# B&R Automation Studio project MotionTestBenchMaster (part 39)

```iecst
xInductionSetupActive	:= TRUE;

CASE uiInductionSetupStep OF
	0:
		IF	VAR_Machine.iq_stParameter.i_uiAxisSelected >= CST_FillerSubModuleHmiStart AND
			VAR_Machine.iq_stParameter.i_uiAxisSelected <= CST_FillerSubModuleHmiStart + CST_LastFillerModuleAxis	THEN

			VAR_Machine.stFillerModule.iq_stParameters.i_uiAxisSelected
				:=	VAR_Machine.iq_stParameter.i_uiAxisSelected - CST_FillerSubModuleHmiStart;

			uiInductionSetupStep	:=	100;
		ELSIF VAR_Machine.iq_stParameter.i_uiAxisSelected >= CST_InletSubModuleHmiStart AND
			VAR_Machine.iq_stParameter.i_uiAxisSelected <= CST_InletSubModuleHmiStart + CST_LastInletModuleAxis THEN

			VAR_Machine.stInletModule.iq_stParameters.i_uiAxisSelected
				:=	VAR_Machine.iq_stParameter.i_uiAxisSelected - CST_InletSubModuleHmiStart;

			uiInductionSetupStep	:=	200;
		ELSIF 	VAR_Machine.iq_stParameter.i_uiAxisSelected >= CST_OutletSubModuleHmiStart AND
			VAR_Machine.iq_stParameter.i_uiAxisSelected <= CST_OutletSubModuleHmiStart + CST_LastOutletModuleAxis THEN

			VAR_Machine.stOutletModule.iq_stParameters.i_uiAxisSelected
				:=	VAR_Machine.iq_stParameter.i_uiAxisSelected - CST_OutletSubModuleHmiStart;

			uiInductionSetupStep	:=	300;
		END_IF

	100:(* Induction motor setup on Filler Module *)
		VAR_Machine.stFillerModule.iq_stCmd.i_xInductionSetup :=	TRUE;

		IF VAR_Machine.stFillerModule.iq_stStatus.q_xInductionSetupActive 	AND
			VAR_Machine.stFillerModule.iq_stStatus.q_xInductionSetupDone	THEN

			VAR_Machine.stFillerModule.iq_stCmd.i_xInductionSetup 			:=	FALSE;
			VAR_Machine.stFillerModule.iq_stParameters.i_uiAxisSelected		:=	CST_FirstFillerModuleAxis;
			uiInductionSetupStep	:=	150;
		END_IF

	150:
		IF NOT VAR_Machine.stFillerModule.iq_stStatus.q_xInductionSetupActive 	AND
			NOT VAR_Machine.stFillerModule.iq_stStatus.q_xInductionSetupDone	THEN
			uiInductionSetupStep	:=	400;
		END_IF

	200:(* Induction motor setup on Inlet Module *)
		VAR_Machine.stInletModule.iq_stCmd.i_xInductionSetup :=	TRUE;

		IF VAR_Machine.stInletModule.iq_stStatus.q_xInductionSetupActive	AND
			VAR_Machine.stInletModule.iq_stStatus.q_xInductionSetupDone	THEN

			VAR_Machine.stInletModule.iq_stCmd.i_xInductionSetup 			:=	FALSE;
			VAR_Machine.stInletModule.iq_stParameters.i_uiAxisSelected		:=	CST_FirstInletModuleAxis;
			uiInductionSetupStep	:=	250;
		END_IF

	250:
		IF NOT VAR_Machine.stInletModule.iq_stStatus.q_xInductionSetupActive 	AND
			NOT	VAR_Machine.stInletModule.iq_stStatus.q_xInductionSetupDone	THEN
			uiInductionSetupStep	:=	400;
		END_IF

	300:(* Induction motor setup on Outlet Module *)
		VAR_Machine.stOutletModule.iq_stCmd.i_xInductionSetup :=	TRUE;

		IF VAR_Machine.stOutletModule.iq_stStatus.q_xInductionSetupActive	AND
			VAR_Machine.stOutletModule.iq_stStatus.q_xInductionSetupDone	THEN

			VAR_Machine.stOutletModule.iq_stCmd.i_xInductionSetup 			:=	FALSE;
			VAR_Machine.stOutletModule.iq_stParameters.i_uiAxisSelected		:=	CST_FirstOutletModuleAxis;
			uiInductionSetupStep	:=	350;
		END_IF

	350:
		IF NOT VAR_Machine.stOutletModule.iq_stStatus.q_xInductionSetupActive	AND
			NOT	VAR_Machine.stOutletModule.iq_stStatus.q_xInductionSetupDone	THEN
			uiInductionSetupStep	:=	400;
		END_IF

	400:
		xInductionSetupDone := TRUE;
END_CASE
END_STEP
ENTRY_ACTION
uiInductionSetupStep	:=	0;
xInductionSetupDone	:=	FALSE;
END_ACTION
EXIT_ACTION
VAR_Machine.stFillerModule.iq_stCmd.i_xInductionSetup 			:=	FALSE;
VAR_Machine.stFillerModule.iq_stParameters.i_uiAxisSelected		:=	CST_FirstFillerModuleAxis;

VAR_Machine.stOutletModule.iq_stCmd.i_xInductionSetup			:=	FALSE;
VAR_Machine.stOutletModule.iq_stParameters.i_uiAxisSelected		:=	CST_FirstOutletModuleAxis;

VAR_Machine.stInletModule.iq_stCmd.i_xInductionSetup			:=	FALSE;
VAR_Machine.stInletModule.iq_stParameters.i_uiAxisSelected		:=	CST_FirstInletModuleAxis;
END_ACTION
TRANSITION FROM InductionSetup TO InductionSetupExit:=
NOT xInductionSetupMode
END_TRANSITION
STEP InductionSetupExit:
xExitStep				:= TRUE;
xInductionSetupDone		:= FALSE;
xInductionSetupActive	:= FALSE;
END_STEP
TRANSITION FROM InductionSetupExit TO ModeSelection:=
xExitStep
END_TRANSITION
(* @SFCISJUMP := 'ModeSelection' *)
TRANSITION FROM ModeSelection TO StepByStep:=
xStepByStepMode
END_TRANSITION
STEP StepByStep:
IF xReactionActive OR uiStepByStep = 140 THEN
	xStepByStepMode	:= FALSE;
END_IF

xStepByStepActive	:= TRUE;

CASE uiStepByStep OF
	0:
		VAR_Machine.stFillerModule.iq_stCmd.i_xAutoMode	:= TRUE;
		VAR_Machine.stInletModule.iq_stCmd.i_xAutoMode	:= VAR_Machine.stInletModule.iq_stStatus.q_xModuleReal;
		VAR_Machine.stOutletModule.iq_stCmd.i_xAutoMode	:= VAR_Machine.stOutletModule.iq_stStatus.q_xModuleReal;
		uiStepByStep	:=	40;

	40:
		IF VAR_Machine.stFillerModule.iq_stStatus.q_xAutoActive		AND
			(VAR_Machine.stInletModule.iq_stStatus.q_xAutoActive	OR NOT
			VAR_Machine.stInletModule.iq_stStatus.q_xModuleReal)	AND
			(VAR_Machine.stOutletModule.iq_stStatus.q_xAutoActive	OR NOT
			VAR_Machine.stOutletModule.iq_stStatus.q_xModuleReal)	THEN

			IF NOT VAR_Machine.stFillerModule.iq_stStatus.q_xSynchroWithOffset	AND
				NOT VAR_Machine.stInletModule.iq_stStatus.q_xSynchroWithOffset	AND
				NOT VAR_Machine.stOutletModule.iq_stStatus.q_xSynchroWithOffset	THEN

				VAR_Machine.stMasterModule.iq_stParameters.i_lrRephasingPosition :=
					FC_RephasingMachine(iq_astInletSubModuleAxis	:= VAR_Machine.stInletModule.iq_astSubModuleAxis,
										iq_astFillerSubModuleAxis	:= VAR_Machine.stFillerModule.iq_astSubModuleAxis,
										iq_astOutletSubModuleAxis	:= VAR_Machine.stOutletModule.iq_astSubModuleAxis);

				VAR_Machine.stFillerModule.iq_stParameters.i_lrRephasingPosition
						:=	VAR_Machine.stMasterModule.iq_stParameters.i_lrRephasingPosition;

				VAR_Machine.stOutletModule.iq_stParameters.i_lrRephasingPosition
						:=	VAR_Machine.stMasterModule.iq_stParameters.i_lrRephasingPosition;

				VAR_Machine.stInletModule.iq_stParameters.i_lrRephasingPosition
					:=	VAR_Machine.stMasterModule.iq_stParameters.i_lrRephasingPosition;

				uiStepByStep	:=	100;
			END_IF
		END_IF

	100:
		VAR_Machine.stMasterModule.iq_stCmd.i_xPositioning				:= TRUE;
		VAR_Machine.stMasterModule.iq_stCmd.i_xMasterRephasingRequest	:= TRUE;

		IF VAR_Machine.stMasterModule.iq_stStatus.q_xPositioningActive AND VAR_Machine.stMasterModule.iq_stStatus.q_xMasterRephased THEN
			VAR_Machine.stMasterModule.iq_stCmd.i_xMasterRephasingRequest	:= FALSE;
			uiStepByStep	:=	110;
		END_IF

	110:
		VAR_Machine.stFillerModule.iq_stCmd.i_xStart	:= TRUE;
		VAR_Machine.stInletModule.iq_stCmd.i_xStart		:= VAR_Machine.stInletModule.iq_stStatus.q_xModuleReal;
		VAR_Machine.stOutletModule.iq_stCmd.i_xStart	:= VAR_Machine.stOutletModule.iq_stStatus.q_xModuleReal;
		uiStepByStep	:=	120;

	120:
		IF VAR_Machine.stFillerModule.iq_stStatus.q_xRealAxesSynchronized		AND
			VAR_Machine.stFillerModule.iq_stStatus.q_xAutoActive				AND
			VAR_Machine.stFillerModule.iq_stStatus.q_xMasterRephased			AND

			((VAR_Machine.stInletModule.iq_stStatus.q_xRealAxesSynchronized		AND
			VAR_Machine.stInletModule.iq_stStatus.q_xMasterRephased				AND
			VAR_Machine.stInletModule.iq_stStatus.q_xAutoActive)				OR NOT
			VAR_Machine.stInletModule.iq_stStatus.q_xModuleReal)				AND

			((VAR_Machine.stOutletModule.iq_stStatus.q_xRealAxesSynchronized	AND
			VAR_Machine.stOutletModule.iq_stStatus.q_xMasterRephased			AND
			VAR_Machine.stOutletModule.iq_stStatus.q_xAutoActive)				OR NOT
			VAR_Machine.stOutletModule.iq_stStatus.q_xModuleReal)				THEN

			VAR_Machine.stMasterModule.iq_stParameters.i_rPositioningOffset
				:= LREAL_TO_REAL(FC_LongRealReminder((VAR_Machine.stMasterModule.iq_stParameters.i_rStopPosition	- VAR_Machine.stMasterModule.iq_astSubModuleAxis[CST_MachineMasterAxis].iq_stStatus.q_stMainAxisStatus.q_lrPosition), 360.0, 0));

			IF VAR_Machine.stMasterModule.iq_stParameters.i_rPositioningOffset > 180.0 THEN
				VAR_Machine.stMasterModule.iq_stParameters.i_rPositioningOffset	:= VAR_Machine.stMasterModule.iq_stParameters.i_rPositioningOffset + 360.0 * (MAX(1, VAR_Machine.iq_stParameter.i_uiNumberOfSteps) - 1);
			ELSE
				VAR_Machine.stMasterModule.iq_stParameters.i_rPositioningOffset	:= VAR_Machine.stMasterModule.iq_stParameters.i_rPositioningOffset + 360.0 * MAX(1, VAR_Machine.iq_stParameter.i_uiNumberOfSteps);
			END_IF

			VAR_Machine.stMasterModule.iq_stCmd.i_xStart	:= TRUE;
			uiStepByStep := 130;
		END_IF

	130:
		IF VAR_Machine.stMasterModule.iq_stStatus.q_xPositioningDone THEN
			VAR_Machine.stMasterModule.iq_stCmd.i_xStart := FALSE;
			uiStepByStep := 140;
		END_IF

	140:

		xStepByStepDone	:= TRUE;
END_CASE
END_STEP
ENTRY_ACTION
uiStepByStep	:= 0;
xStepByStepDone	:= FALSE;
END_ACTION
EXIT_ACTION
VAR_Machine.stFillerModule.iq_stCmd.i_xAutoMode			:= FALSE;
VAR_Machine.stOutletModule.iq_stCmd.i_xAutoMode			:= FALSE;
VAR_Machine.stInletModule.iq_stCmd.i_xAutoMode			:= FALSE;

VAR_Machine.stMasterModule.iq_stCmd.i_xPositioning				:= FALSE;
VAR_Machine.stMasterModule.iq_stCmd.i_xStart					:= FALSE;
VAR_Machine.stMasterModule.iq_stCmd.i_xMasterRephasingRequest	:= FALSE;

VAR_Machine.stFillerModule.iq_stCmd.i_xStart	:= FALSE;
VAR_Machine.stInletModule.iq_stCmd.i_xStart		:= FALSE;
VAR_Machine.stOutletModule.iq_stCmd.i_xStart	:= FALSE;
END_ACTION
TRANSITION FROM StepByStep TO StepExit:=
NOT xStepByStepMode
END_TRANSITION
STEP StepExit:
IF NOT VAR_Machine.stMasterModule.iq_stStatus.q_xPositioningActive	AND
	NOT VAR_Machine.stFillerModule.iq_stStatus.q_xAutoActive		AND

	(NOT VAR_Machine.stOutletModule.iq_stStatus.q_xAutoActive		OR NOT
	VAR_Machine.stOutletModule.iq_stStatus.q_xModuleReal)			AND

	(NOT VAR_Machine.stInletModule.iq_stStatus.q_xAutoActive		OR NOT
	VAR_Machine.stInletModule.iq_stStatus.q_xModuleReal)			AND

	VAR_Machine.iq_stStatus.q_xMachineStopped 						THEN

	xStepByStepDone		:= FALSE;
	xStepByStepActive	:= FALSE;
	xExitStep			:= TRUE;
END_IF
END_STEP
TRANSITION FROM StepExit TO ModeSelection:=
xExitStep
END_TRANSITION
(* @SFCISJUMP := 'ModeSelection' *)
TRANSITION FROM ModeSelection TO StepByStepSingleAxis:=
xStepByStepSingleAxisMode
END_TRANSITION
STEP StepByStepSingleAxis:
xReactionOnFillerModule		:= xReactFillerEmergencyStop 	OR xReactFillerQuickStop		OR xReactFillerStop;//V1.7.2

IF xReactionOnFillerModule OR uiStepByStepSingleAxis = 130 THEN//V1.7.2
	xStepByStepSingleAxisMode	:= FALSE;
END_IF

xStepByStepSingleAxisActive	:= TRUE;

CASE uiStepByStepSingleAxis OF//V4.A.A.1.7.0
	0:
		IF	VAR_Machine.iq_stParameter.i_uiAxisSelected >= CST_FillerSubModuleHmiStart AND
			VAR_Machine.iq_stParameter.i_uiAxisSelected <= CST_FillerSubModuleHmiStart + CST_LastFillerModuleAxis	THEN

			VAR_Machine.stFillerModule.iq_stParameters.i_uiAxisSelected := VAR_Machine.iq_stParameter.i_uiAxisSelected - CST_FillerSubModuleHmiStart;

			uiStepByStepSingleAxis	:=	100;//Filler Module
		ELSIF VAR_Machine.iq_stParameter.i_uiAxisSelected >= CST_InletSubModuleHmiStart AND
			VAR_Machine.iq_stParameter.i_uiAxisSelected <= CST_InletSubModuleHmiStart + CST_LastInletModuleAxis THEN

			VAR_Machine.stInletModule.iq_stParameters.i_uiAxisSelected := VAR_Machine.iq_stParameter.i_uiAxisSelected - CST_InletSubModuleHmiStart;

			uiStepByStepSingleAxis	:=	200;//Inlet Module
		ELSIF 	VAR_Machine.iq_stParameter.i_uiAxisSelected >= CST_OutletSubModuleHmiStart AND
			VAR_Machine.iq_stParameter.i_uiAxisSelected <= CST_OutletSubModuleHmiStart + CST_LastOutletModuleAxis THEN

			VAR_Machine.stOutletModule.iq_stParameters.i_uiAxisSelected := VAR_Machine.iq_stParameter.i_uiAxisSelected - CST_OutletSubModuleHmiStart;

			uiStepByStepSingleAxis	:=	300;//Outlet module
		ELSIF VAR_Machine.iq_stParameter.i_uiAxisSelected = CST_MachinePhasingOffset THEN
			uiStepByStepSingleAxis	:=	700;
		END_IF

	100:

		VAR_Machine.stFillerModule.iq_stParameters.i_rPositioningOffset
						:= LREAL_TO_REAL(FC_LongRealReminder((VAR_Machine.stFillerModule.iq_stParameters.i_rStopPosition	- VAR_Machine.stFillerModule.iq_astSubModuleAxis[VAR_Machine.stFillerModule.iq_stParameters.i_uiAxisSelected].iq_stStatus.q_stMainAxisStatus.q_lrPosition), 360.0, 0));

		IF VAR_Machine.stFillerModule.iq_stParameters.i_rPositioningOffset > 180.0 THEN
			VAR_Machine.stFillerModule.iq_stParameters.i_rPositioningOffset	:= VAR_Machine.stFillerModule.iq_stParameters.i_rPositioningOffset + 360.0 * (MAX(1, VAR_Machine.iq_stParameter.i_uiNumberOfSteps) - 1);
		ELSE
			VAR_Machine.stFillerModule.iq_stParameters.i_rPositioningOffset	:= VAR_Machine.stFillerModule.iq_stParameters.i_rPositioningOffset + 360.0 * MAX(1, VAR_Machine.iq_stParameter.i_uiNumberOfSteps);
		END_IF

		uiStepByStepSingleAxis := 110;

	110://
		VAR_Machine.stFillerModule.iq_stCmd.i_xPositioningMode			:= TRUE;
		VAR_Machine.stFillerModule.iq_stCmd.i_xStepByStepSingleAxis		:= TRUE;

		IF VAR_Machine.stFillerModule.iq_stStatus.q_xPositioningActive 	AND
			VAR_Machine.stFillerModule.iq_stStatus.q_xPositioningDone	THEN

			VAR_Machine.stFillerModule.iq_stCmd.i_xPositioningMode 			:=	FALSE;
			VAR_Machine.stFillerModule.iq_stCmd.i_xStepByStepSingleAxis		:= FALSE;
			VAR_Machine.stFillerModule.iq_stParameters.i_rPositioningOffset	:=	0.0;
			uiStepByStepSingleAxis	:=	120;
		END_IF

	120:
		IF NOT VAR_Machine.stFillerModule.iq_stStatus.q_xPositioningActive 	AND
			NOT VAR_Machine.stFillerModule.iq_stStatus.q_xPositioningDone	THEN
			uiStepByStepSingleAxis	:=	130;
		END_IF

	130:
		xStepByStepSingleAxisDone	:= TRUE;

END_CASE
END_STEP
ENTRY_ACTION
uiStepByStepSingleAxis		:= 0;
xStepByStepSingleAxisDone	:= FALSE;
xReactionOnFillerModule		:= FALSE;//V1.7.2
END_ACTION
EXIT_ACTION
VAR_Machine.stFillerModule.iq_stCmd.i_xPositioningMode 			:= FALSE;
VAR_Machine.stFillerModule.iq_stCmd.i_xStart					:= FALSE;	//v1.2
VAR_Machine.stFillerModule.iq_stParameters.i_rPositioningOffset	:= 0.0;
VAR_Machine.stFillerModule.iq_stParameters.i_uiAxisSelected		:= CST_FirstFillerModuleAxis;
VAR_Machine.stFillerModule.iq_stCmd.i_xAutoMode					:= FALSE;

VAR_Machine.stOutletModule.iq_stCmd.i_xPositioningMode			:= FALSE;
VAR_Machine.stOutletModule.iq_stCmd.i_xStart					:= FALSE;	//v1.2
VAR_Machine.stOutletModule.iq_stParameters.i_rPositioningOffset	:= 0.0;
VAR_Machine.stOutletModule.iq_stParameters.i_uiAxisSelected		:= CST_FirstOutletModuleAxis;
VAR_Machine.stOutletModule.iq_stCmd.i_xAutoMode					:= FALSE;

VAR_Machine.stInletModule.iq_stCmd.i_xPositioningMode			:= FALSE;
VAR_Machine.stInletModule.iq_stCmd.i_xStart						:= FALSE;	//v1.2
VAR_Machine.stInletModule.iq_stParameters.i_rPositioningOffset	:= 0.0;
VAR_Machine.stInletModule.iq_stParameters.i_uiAxisSelected		:= CST_FirstInletModuleAxis;
VAR_Machine.stInletModule.iq_stCmd.i_xAutoMode					:= FALSE;

VAR_Machine.stFillerModule.iq_stCmd.i_xStepByStepSingleAxis		:= FALSE;
END_ACTION
TRANSITION FROM StepByStepSingleAxis TO StepSingleAxisExit:=
NOT xStepByStepSingleAxisMode
END_TRANSITION
STEP StepSingleAxisExit:
xExitStep						:= 	TRUE;
xStepByStepSingleAxisDone		:=	FALSE;
xStepByStepSingleAxisActive		:=	FALSE;
END_STEP
TRANSITION FROM StepSingleAxisExit TO ModeSelection:=
xExitStep
END_TRANSITION
(* @SFCISJUMP := 'ModeSelection' *)
TRANSITION FROM ModeSelection TO StepByStepSingleAxisRev:=
xStepByStepSingleAxisReverseMode
END_TRANSITION
STEP StepByStepSingleAxisRev:
xReactionOnFillerModule		:= xReactFillerEmergencyStop 	OR xReactFillerQuickStop		OR xReactFillerStop;//V1.7.2

IF xReactionOnFillerModule OR uiStepByStepSingleReverseAxis = 130 THEN//V1.7.2
	xStepByStepSingleAxisReverseMode	:= FALSE;
END_IF

xStepByStepSingleAxisRevActive	:= TRUE;

CASE uiStepByStepSingleReverseAxis OF//V4.A.A.1.7.0
	0:
		IF	VAR_Machine.iq_stParameter.i_uiAxisSelected >= CST_FillerSubModuleHmiStart AND
			VAR_Machine.iq_stParameter.i_uiAxisSelected <= CST_FillerSubModuleHmiStart + CST_LastFillerModuleAxis	THEN

			VAR_Machine.stFillerModule.iq_stParameters.i_uiAxisSelected := VAR_Machine.iq_stParameter.i_uiAxisSelected - CST_FillerSubModuleHmiStart;

			uiStepByStepSingleReverseAxis	:=	100;//Filler Module
		ELSIF VAR_Machine.iq_stParameter.i_uiAxisSelected >= CST_InletSubModuleHmiStart AND
			VAR_Machine.iq_stParameter.i_uiAxisSelected <= CST_InletSubModuleHmiStart + CST_LastInletModuleAxis THEN

			VAR_Machine.stInletModule.iq_stParameters.i_uiAxisSelected := VAR_Machine.iq_stParameter.i_uiAxisSelected - CST_InletSubModuleHmiStart;

			uiStepByStepSingleReverseAxis	:=	200;//Inlet Module
		ELSIF 	VAR_Machine.iq_stParameter.i_uiAxisSelected >= CST_OutletSubModuleHmiStart AND
			VAR_Machine.iq_stParameter.i_uiAxisSelected <= CST_OutletSubModuleHmiStart + CST_LastOutletModuleAxis THEN

			VAR_Machine.stOutletModule.iq_stParameters.i_uiAxisSelected := VAR_Machine.iq_stParameter.i_uiAxisSelected - CST_OutletSubModuleHmiStart;

			uiStepByStepSingleReverseAxis	:=	300;//Outlet module
		ELSIF VAR_Machine.iq_stParameter.i_uiAxisSelected = CST_MachinePhasingOffset THEN
			uiStepByStepSingleReverseAxis	:=	700;
		END_IF

	100:

		VAR_Machine.stFillerModule.iq_stParameters.i_rPositioningOffset
		:= LREAL_TO_REAL(FC_LongRealReminder((VAR_Machine.stFillerModule.iq_stParameters.i_rStopPosition	- VAR_Machine.stFillerModule.iq_astSubModuleAxis[VAR_Machine.stFillerModule.iq_stParameters.i_uiAxisSelected].iq_stStatus.q_stMainAxisStatus.q_lrPosition), 360.0, 0));

		IF VAR_Machine.stFillerModule.iq_stParameters.i_rPositioningOffset > 180.0 THEN
			VAR_Machine.stFillerModule.iq_stParameters.i_rPositioningOffset	:= -(VAR_Machine.stFillerModule.iq_stParameters.i_rPositioningOffset + 360.0 * (MAX(1, VAR_Machine.iq_stParameter.i_uiNumberOfSteps) - 1));
		ELSE
			VAR_Machine.stFillerModule.iq_stParameters.i_rPositioningOffset	:= -(VAR_Machine.stFillerModule.iq_stParameters.i_rPositioningOffset + 360.0 * MAX(1, VAR_Machine.iq_stParameter.i_uiNumberOfSteps));
		END_IF

		uiStepByStepSingleReverseAxis := 110;

	110://
		VAR_Machine.stFillerModule.iq_stCmd.i_xPositioningMode			:= TRUE;
		VAR_Machine.stFillerModule.iq_stCmd.i_xStepByStepSingleAxis		:= TRUE;

		IF VAR_Machine.stFillerModule.iq_stStatus.q_xPositioningActive 	AND
			VAR_Machine.stFillerModule.iq_stStatus.q_xPositioningDone	THEN

			VAR_Machine.stFillerModule.iq_stCmd.i_xPositioningMode 			:=	FALSE;
			VAR_Machine.stFillerModule.iq_stCmd.i_xStepByStepSingleAxis		:= FALSE;
			VAR_Machine.stFillerModule.iq_stParameters.i_rPositioningOffset	:=	0.0;
			uiStepByStepSingleReverseAxis	:=	120;
		END_IF

	120:
		IF NOT VAR_Machine.stFillerModule.iq_stStatus.q_xPositioningActive 	AND
			NOT VAR_Machine.stFillerModule.iq_stStatus.q_xPositioningDone	THEN
			uiStepByStepSingleReverseAxis	:=	130;
		END_IF

	130:
		xStepByStepSingleAxisReverseDone	:= TRUE;

END_CASE
END_STEP
ENTRY_ACTION
uiStepByStepSingleReverseAxis		:= 0;
xStepByStepSingleAxisReverseDone	:= FALSE;//v999
xReactionOnFillerModule				:= FALSE;
END_ACTION
EXIT_ACTION
VAR_Machine.stFillerModule.iq_stCmd.i_xPositioningMode 			:= FALSE;
VAR_Machine.stFillerModule.iq_stCmd.i_xStart					:= FALSE;	//v1.2
VAR_Machine.stFillerModule.iq_stParameters.i_rPositioningOffset	:= 0.0;
VAR_Machine.stFillerModule.iq_stParameters.i_uiAxisSelected		:= CST_FirstFillerModuleAxis;
VAR_Machine.stFillerModule.iq_stCmd.i_xAutoMode					:= FALSE;

VAR_Machine.stOutletModule.iq_stCmd.i_xPositioningMode			:= FALSE;
VAR_Machine.stOutletModule.iq_stCmd.i_xStart					:= FALSE;	//v1.2
VAR_Machine.stOutletModule.iq_stParameters.i_rPositioningOffset	:= 0.0;
VAR_Machine.stOutletModule.iq_stParameters.i_uiAxisSelected		:= CST_FirstOutletModuleAxis;
VAR_Machine.stOutletModule.iq_stCmd.i_xAutoMode					:= FALSE;

VAR_Machine.stInletModule.iq_stCmd.i_xPositioningMode			:= FALSE;
VAR_Machine.stInletModule.iq_stCmd.i_xStart						:= FALSE;	//v1.2
VAR_Machine.stInletModule.iq_stParameters.i_rPositioningOffset	:= 0.0;
VAR_Machine.stInletModule.iq_stParameters.i_uiAxisSelected		:= CST_FirstInletModuleAxis;
VAR_Machine.stInletModule.iq_stCmd.i_xAutoMode					:= FALSE;

VAR_Machine.stFillerModule.iq_stCmd.i_xStepByStepSingleAxis		:= FALSE;
END_ACTION
TRANSITION FROM StepByStepSingleAxisRev TO StepByStepSingleAxisRevExit:=
NOT xStepByStepSingleAxisReverseMode
END_TRANSITION
STEP StepByStepSingleAxisRevExit:
xExitStep						:= 	TRUE;
xStepByStepSingleAxisReverseDone		:=	FALSE;
xStepByStepSingleAxisRevActive		:=	FALSE;
END_STEP
TRANSITION FROM StepByStepSingleAxisRevExit TO ModeSelection:=
xExitStep
END_TRANSITION
(* @SFCISJUMP := 'ModeSelection' *)
STEP Auto:
IF xReactionActive OR NOT xInputAuto THEN
	xAutoMode	:= FALSE;
END_IF

xAutoActive	:= TRUE;

CASE uiAutoStep OF
	0:
		VAR_Machine.stFillerModule.iq_stCmd.i_xAutoMode	:=	TRUE;
		VAR_Machine.stOutletModule.iq_stCmd.i_xAutoMode	:=	VAR_Machine.stOutletModule.iq_stStatus.q_xModuleReal;
		VAR_Machine.stInletModule.iq_stCmd.i_xAutoMode	:=	VAR_Machine.stInletModule.iq_stStatus.q_xModuleReal;

		uiAutoStep	:= 40;

	40:
		IF 	VAR_Machine.stFillerModule.iq_stStatus.q_xAutoActive	AND
			(VAR_Machine.stOutletModule.iq_stStatus.q_xAutoActive	OR NOT
			VAR_Machine.stOutletModule.iq_stStatus.q_xModuleReal)	AND
			(VAR_Machine.stInletModule.iq_stStatus.q_xAutoActive	OR NOT
			VAR_Machine.stInletModule.iq_stStatus.q_xModuleReal)	THEN

			IF 	NOT VAR_Machine.stFillerModule.iq_stStatus.q_xSynchroWithOffset		AND
				NOT VAR_Machine.stOutletModule.iq_stStatus.q_xSynchroWithOffset		AND
				NOT VAR_Machine.stInletModule.iq_stStatus.q_xSynchroWithOffset		THEN

				VAR_Machine.stMasterModule.iq_stParameters.i_lrRephasingPosition	:=
				FC_RephasingMachine(iq_astInletSubModuleAxis	:=	VAR_Machine.stInletModule.iq_astSubModuleAxis,
									iq_astFillerSubModuleAxis	:=	VAR_Machine.stFillerModule.iq_astSubModuleAxis,
									iq_astOutletSubModuleAxis	:=	VAR_Machine.stOutletModule.iq_astSubModuleAxis);

				VAR_Machine.stFillerModule.iq_stParameters.i_lrRephasingPosition
					:=	VAR_Machine.stMasterModule.iq_stParameters.i_lrRephasingPosition;

				VAR_Machine.stOutletModule.iq_stParameters.i_lrRephasingPosition
					:=	VAR_Machine.stMasterModule.iq_stParameters.i_lrRephasingPosition;

				VAR_Machine.stInletModule.iq_stParameters.i_lrRephasingPosition
					:=	VAR_Machine.stMasterModule.iq_stParameters.i_lrRephasingPosition;

				uiAutoStep	:= 100;
			END_IF
		END_IF

	100:(* Wait Master Rephased *)
		VAR_Machine.stMasterModule.iq_stCmd.i_xAutoMode					:=	TRUE;
		VAR_Machine.stMasterModule.iq_stCmd.i_xMasterRephasingRequest	:= 	TRUE;

		IF VAR_Machine.stMasterModule.iq_stStatus.q_xAutoActive AND VAR_Machine.stMasterModule.iq_stStatus.q_xMasterRephased THEN
			VAR_Machine.stMasterModule.iq_stCmd.i_xMasterRephasingRequest	:= 	FALSE;
			uiAutoStep	:= 110;
		END_IF

	110:(* Wait for start Signal *)
		IF VAR_Machine.iq_stCmd.i_xStart THEN
			VAR_Machine.stFillerModule.iq_stCmd.i_xStart	:=	TRUE;
			VAR_Machine.stOutletModule.iq_stCmd.i_xStart	:=	VAR_Machine.stOutletModule.iq_stStatus.q_xModuleReal;
			VAR_Machine.stInletModule.iq_stCmd.i_xStart		:=	VAR_Machine.stInletModule.iq_stStatus.q_xModuleReal;
			uiAutoStep	:= 120;
		END_IF

	120:(* Wait for submodules synchronized *)
		IF VAR_Machine.stFillerModule.iq_stStatus.q_xRealAxesSynchronized		AND
				VAR_Machine.stFillerModule.iq_stStatus.q_xAutoActive			AND
				VAR_Machine.stFillerModule.iq_stStatus.q_xMasterRephased		AND

			((VAR_Machine.stOutletModule.iq_stStatus.q_xRealAxesSynchronized	AND
				VAR_Machine.stOutletModule.iq_stStatus.q_xMasterRephased		AND
				VAR_Machine.stOutletModule.iq_stStatus.q_xAutoActive)			OR NOT
				VAR_Machine.stOutletModule.iq_stStatus.q_xModuleReal)			AND

			((VAR_Machine.stInletModule.iq_stStatus.q_xRealAxesSynchronized		AND
				VAR_Machine.stInletModule.iq_stStatus.q_xMasterRephased			AND
				VAR_Machine.stInletModule.iq_stStatus.q_xAutoActive)			OR NOT
				VAR_Machine.stInletModule.iq_stStatus.q_xModuleReal)			THEN

			VAR_Machine.stMasterModule.iq_stCmd.i_xStart	:= TRUE;
			xEncEmulationEnable	:= TRUE;
			uiAutoStep	:= 140;
		END_IF

	140:
		IF NOT VAR_Machine.iq_stCmd.i_xStart THEN
			VAR_Machine.stMasterModule.iq_stCmd.i_xStart	:= FALSE;
			uiAutoStep	:= 150;
		ELSIF VAR_Machine.iq_stCmd.i_xAxisPhaseShift THEN
			IF 	VAR_Machine.iq_stParameter.i_uiAxisSelected >= CST_FillerSubModuleHmiStart AND
				VAR_Machine.iq_stParameter.i_uiAxisSelected <= CST_FillerSubModuleHmiStart + CST_LastFillerModuleAxis	THEN

				VAR_Machine.stFillerModule.iq_stParameters.i_uiAxisSelected
					:=	VAR_Machine.iq_stParameter.i_uiAxisSelected - CST_FillerSubModuleHmiStart;

				VAR_Machine.stFillerModule.iq_stParameters.i_rPhaseShiftDistance
					:=	LREAL_TO_REAL(FC_TeensOfmmToDegrees(VAR_Machine.iq_stParameter.i_iAxisPhaseShiftDistance, CFG_MC.Mechanical.MachineStep, TRUE, FALSE));

				uiAutoStep	:= 200;
			ELSIF 	VAR_Machine.iq_stParameter.i_uiAxisSelected >= CST_OutletSubModuleHmiStart AND
				VAR_Machine.iq_stParameter.i_uiAxisSelected <= CST_OutletSubModuleHmiStart + CST_LastOutletModuleAxis	THEN

				VAR_Machine.stOutletModule.iq_stParameters.i_uiAxisSelected
					:=	VAR_Machine.iq_stParameter.i_uiAxisSelected - CST_OutletSubModuleHmiStart;

				VAR_Machine.stOutletModule.iq_stParameters.i_rPhaseShiftDistance
					:=	LREAL_TO_REAL(FC_TeensOfmmToDegrees(VAR_Machine.iq_stParameter.i_iAxisPhaseShiftDistance, CFG_MC.Mechanical.MachineStep, TRUE, FALSE));

				uiAutoStep	:= 300;
			ELSIF 	VAR_Machine.iq_stParameter.i_uiAxisSelected >= CST_InletSubModuleHmiStart AND
				VAR_Machine.iq_stParameter.i_uiAxisSelected <= CST_InletSubModuleHmiStart + CST_LastInletModuleAxis		THEN

				VAR_Machine.stInletModule.iq_stParameters.i_uiAxisSelected
					:=	VAR_Machine.iq_stParameter.i_uiAxisSelected - CST_InletSubModuleHmiStart;

				VAR_Machine.stInletModule.iq_stParameters.i_rPhaseShiftDistance
					:=	LREAL_TO_REAL(FC_TeensOfmmToDegrees(VAR_Machine.iq_stParameter.i_iAxisPhaseShiftDistance, CFG_MC.Mechanical.MachineStep, TRUE, FALSE));

				uiAutoStep	:= 400;
			END_IF
		END_IF

	150:
		IF VAR_Machine.stMasterModule.iq_stStatus.q_xModuleStopped THEN
			xEncEmulationEnable	:= FALSE;
			uiAutoStep	:=	160;
		END_IF

	160:
		IF VAR_Machine.iq_stCmd.i_xStart THEN
			VAR_Machine.stMasterModule.iq_stCmd.i_xStart	:= TRUE;
			xEncEmulationEnable	:= TRUE;
			uiAutoStep	:= 140;
		ELSIF VAR_Machine.stMasterModule.iq_stStatus.q_xSynchroWithOffset		OR
				VAR_Machine.stFillerModule.iq_stStatus.q_xSynchroWithOffset		OR
				(VAR_Machine.stOutletModule.iq_stStatus.q_xSynchroWithOffset	AND
				VAR_Machine.stOutletModule.iq_stStatus.q_xModuleReal)			OR
				(VAR_Machine.stInletModule.iq_stStatus.q_xSynchroWithOffset		AND
				VAR_Machine.stInletModule.iq_stStatus.q_xModuleReal)			THEN
			uiAutoStep	:= 800;
		END_IF

	200:
		VAR_Machine.stFillerModule.iq_stCmd.i_xPhaseShift	:= TRUE;
		uiAutoStep	:= 210;

	210:
		IF VAR_Machine.stFillerModule.iq_stStatus.q_xPhaseShiftDone AND NOT VAR_Machine.iq_stCmd.i_xAxisPhaseShift THEN
			VAR_Machine.stFillerModule.iq_stCmd.i_xPhaseShift	:= FALSE;
			xEncEmulationEnable	:= TRUE;
			uiAutoStep	:= 140;
		END_IF

	300:
		VAR_Machine.stOutletModule.iq_stCmd.i_xPhaseShift	:= TRUE;
		uiAutoStep	:= 310;

	310:
		IF VAR_Machine.stOutletModule.iq_stStatus.q_xPhaseShiftDone AND NOT VAR_Machine.iq_stCmd.i_xAxisPhaseShift THEN
			VAR_Machine.stOutletModule.iq_stCmd.i_xPhaseShift	:= FALSE;
			xEncEmulationEnable	:= TRUE;
			uiAutoStep	:= 140;
		END_IF

	400:
		VAR_Machine.stInletModule.iq_stCmd.i_xPhaseShift	:= TRUE;
		uiAutoStep	:= 410;

	410:
		IF VAR_Machine.stInletModule.iq_stStatus.q_xPhaseShiftDone AND NOT VAR_Machine.iq_stCmd.i_xAxisPhaseShift THEN
			VAR_Machine.stInletModule.iq_stCmd.i_xPhaseShift	:= FALSE;
			xEncEmulationEnable	:= TRUE;
			uiAutoStep	:= 140;
		END_IF

	800:
		VAR_Machine.stMasterModule.iq_stCmd.i_xPhaseCompensation	:= VAR_Machine.stMasterModule.iq_stStatus.q_xSynchroWithOffset;
		VAR_Machine.stFillerModule.iq_stCmd.i_xPhaseCompensation	:= VAR_Machine.stFillerModule.iq_stStatus.q_xSynchroWithOffset;
		VAR_Machine.stInletModule.iq_stCmd.i_xPhaseCompensation		:= VAR_Machine.stInletModule.iq_stStatus.q_xSynchroWithOffset;
		VAR_Machine.stOutletModule.iq_stCmd.i_xPhaseCompensation	:= VAR_Machine.stOutletModule.iq_stStatus.q_xSynchroWithOffset;

		uiAutoStep	:= 810;

	810:
		IF NOT VAR_Machine.stMasterModule.iq_stStatus.q_xSynchroWithOffset		AND
			NOT VAR_Machine.stFillerModule.iq_stStatus.q_xSynchroWithOffset		AND
			(NOT VAR_Machine.stInletModule.iq_stStatus.q_xSynchroWithOffset		OR
			NOT VAR_Machine.stInletModule.iq_stStatus.q_xModuleReal)			AND
		   (NOT VAR_Machine.stOutletModule.iq_stStatus.q_xSynchroWithOffset		OR
			NOT VAR_Machine.stOutletModule.iq_stStatus.q_xModuleReal)			THEN

			VAR_Machine.stMasterModule.iq_stCmd.i_xPhaseCompensation	:= FALSE;
			VAR_Machine.stFillerModule.iq_stCmd.i_xPhaseCompensation	:= FALSE;
			VAR_Machine.stInletModule.iq_stCmd.i_xPhaseCompensation		:= FALSE;
			VAR_Machine.stOutletModule.iq_stCmd.i_xPhaseCompensation	:= FALSE;

			xEncEmulationEnable	:= TRUE;
			uiAutoStep	:= 140;
		END_IF
END_CASE
END_STEP
ENTRY_ACTION
uiAutoStep	:=	0;
END_ACTION
TRANSITION FROM Auto TO AutoExit:=
NOT xAutoMode
END_TRANSITION
STEP AutoExit:
IF	NOT VAR_Machine.stMasterModule.iq_stStatus.q_xAutoActive	AND
	NOT VAR_Machine.stFillerModule.iq_stStatus.q_xAutoActive	AND
	(NOT VAR_Machine.stInletModule.iq_stStatus.q_xAutoActive	OR NOT
	VAR_Machine.stInletModule.iq_stStatus.q_xModuleReal)		AND
	(NOT VAR_Machine.stOutletModule.iq_stStatus.q_xAutoActive	OR NOT
	VAR_Machine.stOutletModule.iq_stStatus.q_xModuleReal)		THEN

	xExitStep	:= TRUE;
END_IF
END_STEP
ENTRY_ACTION
VAR_Machine.stFillerModule.iq_stCmd.i_xPhaseShift	:= FALSE;
VAR_Machine.stOutletModule.iq_stCmd.i_xPhaseShift	:= FALSE;
VAR_Machine.stInletModule.iq_stCmd.i_xPhaseShift	:= FALSE;

VAR_Machine.stMasterModule.iq_stCmd.i_xStart	:= FALSE;
VAR_Machine.stFillerModule.iq_stCmd.i_xStart	:= FALSE;
VAR_Machine.stOutletModule.iq_stCmd.i_xStart	:= FALSE;
VAR_Machine.stInletModule.iq_stCmd.i_xStart		:= FALSE;

VAR_Machine.stMasterModule.iq_stCmd.i_xAutoMode	:= FALSE;
VAR_Machine.stFillerModule.iq_stCmd.i_xAutoMode	:= FALSE;
VAR_Machine.stOutletModule.iq_stCmd.i_xAutoMode	:= FALSE;
VAR_Machine.stInletModule.iq_stCmd.i_xAutoMode	:= FALSE;

VAR_Machine.stMasterModule.iq_stCmd.i_xMasterRephasingRequest	:= FALSE;

VAR_Machine.stMasterModule.iq_stCmd.i_xPhaseCompensation	:= FALSE;
VAR_Machine.stFillerModule.iq_stCmd.i_xPhaseCompensation	:= FALSE;
VAR_Machine.stOutletModule.iq_stCmd.i_xPhaseCompensation	:= FALSE;
VAR_Machine.stInletModule.iq_stCmd.i_xPhaseCompensation		:= FALSE;

xEncEmulationEnable	:= FALSE;
END_ACTION
TRANSITION FROM AutoExit TO ModeSelection:=
xExitStep
END_TRANSITION
(* @SFCISJUMP := 'ModeSelection' *)
STEP SetException:
xEnableMpAlarmXCore := VAR_Machine.stMasterModule.iq_stStatus.q_xAlarmXCoreEnabled		AND
						(VAR_Machine.stFillerModule.iq_stStatus.q_xAlarmXCoreEnabled	AND (VAR_Machine.stFillerModule.iq_stStatus.q_xModuleReal	OR	VAR_Machine.stFillerModule.iq_stStatus.q_xInitDone))	AND
						(VAR_Machine.stInletModule.iq_stStatus.q_xAlarmXCoreEnabled		AND (VAR_Machine.stInletModule.iq_stStatus.q_xModuleReal	OR	VAR_Machine.stInletModule.iq_stStatus.q_xInitDone))		AND
						(VAR_Machine.stOutletModule.iq_stStatus.q_xAlarmXCoreEnabled	AND (VAR_Machine.stOutletModule.iq_stStatus.q_xModuleReal	OR	VAR_Machine.stOutletModule.iq_stStatus.q_xInitDone));

fbMpAlarmXCore(MpLink := ADR(gMainAlarmXCoreLink), Enable := xEnableMpAlarmXCore);

VAR_Machine.stMasterModule.iq_stCmd.i_xAlarmInitOk	:=	fbMpAlarmXCore.Active;
VAR_Machine.stFillerModule.iq_stCmd.i_xAlarmInitOk	:=	fbMpAlarmXCore.Active;
VAR_Machine.stInletModule.iq_stCmd.i_xAlarmInitOk	:=	fbMpAlarmXCore.Active;
VAR_Machine.stOutletModule.iq_stCmd.i_xAlarmInitOk	:=	fbMpAlarmXCore.Active;

(* Alarm *)
fbQuickStopFromPlc(i_xConditions :=  NOT  xInputMulti AND NOT VAR_Machine.iq_stCmd.i_xQuickStop);

(* Read reactions *)
xReactionMachineQuickStop	:= MpAlarmXCheckReaction(MpLink := gMainAlarmXCoreLink, Name := 'MachineQuickStop');

xReactMasterStop			:= MpAlarmXCheckReaction(MpLink := gMainAlarmXCoreLink, Name := 'MasterStop');
xReactMasterQuickStop		:= MpAlarmXCheckReaction(MpLink := gMainAlarmXCoreLink, Name := 'MasterQuickStop');
xReactMasterShutdown		:= MpAlarmXCheckReaction(MpLink := gMainAlarmXCoreLink, Name := 'MasterShutdown');

xReactFillerStop			:= MpAlarmXCheckReaction(MpLink := gMainAlarmXCoreLink, Name := 'FillerStop');
xReactFillerQuickStop		:= MpAlarmXCheckReaction(MpLink := gMainAlarmXCoreLink, Name := 'FillerQuickStop');
xReactFillerEmergencyStop	:= MpAlarmXCheckReaction(MpLink := gMainAlarmXCoreLink, Name := 'FillerEmergencyStop');

xReactInletStop				:= MpAlarmXCheckReaction(MpLink := gMainAlarmXCoreLink, Name := 'InletStop');
xReactInletQuickStop		:= MpAlarmXCheckReaction(MpLink := gMainAlarmXCoreLink, Name := 'InletQuickStop');
xReactInletEmergencyStop	:= MpAlarmXCheckReaction(MpLink := gMainAlarmXCoreLink, Name := 'InletEmergencyStop');

xReactOutletStop			:= MpAlarmXCheckReaction(MpLink := gMainAlarmXCoreLink, Name := 'OutletStop');
xReactOutletQuickStop		:= MpAlarmXCheckReaction(MpLink := gMainAlarmXCoreLink, Name := 'OutletQuickStop');
xReactOutletEmergencyStop	:= MpAlarmXCheckReaction(MpLink := gMainAlarmXCoreLink, Name := 'OutletEmergencyStop');

(* Check if reaction is ready to be performed *)
xReactionReadyToBePerformed	:= CFG_MC.Generic.DisengageImmediately			OR
								NOT xCombiActive 							OR
								VAR_Machine.iq_stStatus.q_xMachineStopped	OR
								(VAR_Machine.iq_stCmd.i_xOkToDisengage		AND
								(xReactMasterShutdown));

IF NOT xReactionReadyToBePerformed THEN
	xReactionMachineQuickStop	:= FALSE;

	xReactMasterStop			:= FALSE;
	xReactMasterQuickStop		:= FALSE;
	xReactMasterShutdown		:= FALSE;

	xReactFillerStop			:= FALSE;
	xReactFillerQuickStop		:= FALSE;
	xReactFillerEmergencyStop	:= FALSE;

	xReactInletStop				:= FALSE;
	xReactInletQuickStop		:= FALSE;
	xReactInletEmergencyStop	:= FALSE;

	xReactOutletStop			:= FALSE;
	xReactOutletQuickStop		:= FALSE;
	xReactOutletEmergencyStop	:= FALSE;
END_IF

(***** SHUTDOWN *****)
VAR_Machine.stMasterModule.iq_stCmd.i_xShutdown			:= xReactMasterShutdown;
VAR_Machine.stFillerModule.iq_stCmd.i_xShutdown			:= xReactMasterShutdown;
VAR_Machine.stInletModule.iq_stCmd.i_xShutdown			:= xReactMasterShutdown;
VAR_Machine.stOutletModule.iq_stCmd.i_xShutdown			:= xReactMasterShutdown;

(***** EMERGENCY STOP REACTION *****)
VAR_Machine.stMasterModule.iq_stCmd.i_xEmergencyStop	:= (xReactFillerEmergencyStop OR xReactInletEmergencyStop OR xReactOutletEmergencyStop);
VAR_Machine.stFillerModule.iq_stCmd.i_xEmergencyStop	:= xReactFillerEmergencyStop;
VAR_Machine.stInletModule.iq_stCmd.i_xEmergencyStop		:= xReactInletEmergencyStop;
VAR_Machine.stOutletModule.iq_stCmd.i_xEmergencyStop	:= xReactOutletEmergencyStop;

(***** QUICK STOP *****)
VAR_Machine.stMasterModule.iq_stCmd.i_xQuickStop		:= (xReactMasterQuickStop OR xReactFillerQuickStop OR xReactInletQuickStop OR xReactOutletQuickStop OR xReactionMachineQuickStop);
VAR_Machine.stFillerModule.iq_stCmd.i_xQuickStop		:= xReactFillerQuickStop;
VAR_Machine.stInletModule.iq_stCmd.i_xQuickStop			:= xReactInletQuickStop;
VAR_Machine.stOutletModule.iq_stCmd.i_xQuickStop		:= xReactOutletQuickStop;

(***** IN PHASE STOP *****)
VAR_Machine.stMasterModule.iq_stCmd.i_xInPhaseStop		:= (xReactMasterStop OR xReactFillerStop OR xReactInletStop OR xReactOutletStop);
VAR_Machine.stFillerModule.iq_stCmd.i_xInPhaseStop		:= xReactFillerStop;
VAR_Machine.stInletModule.iq_stCmd.i_xInPhaseStop		:= xReactInletStop;
VAR_Machine.stOutletModule.iq_stCmd.i_xInPhaseStop		:= xReactOutletStop;

xReactionActive	:= xReactMasterShutdown			OR
					(xReactFillerEmergencyStop 	OR xReactInletEmergencyStop		OR xReactOutletEmergencyStop)	OR
					(xReactionMachineQuickStop	OR xReactMasterQuickStop 		OR xReactFillerQuickStop 		OR xReactInletQuickStop	OR xReactOutletQuickStop);

tofReactionActive(IN := xReactionActive, PT:= T#1s);

tonFanSeamerActive(IN := MC_InputOutput.Network.Machine.Commands.FanSeamerOn, PT := t#3s);
fbSeamerFanFault(i_xConditions	:= CFG_Par.Motors.CoolingFan.Outlet.Main.Present				AND (NOT MC_InputOutput.Network.Machine.Commands.FanSeamerThermalOverload OR
									(NOT MC_InputOutput.Network.Machine.Commands.FanSeamerOn	AND MC_InputOutput.Network.Outlet.Status.ModuleRunning) OR
									(tonFanSeamerActive.Q	AND MC_InputOutput.Network.Machine.Commands.FanSeamerFeedback)));

MC_InputOutput.Network.Machine.Exceptions.FanSeamearFault		:= fbSeamerFanFault.q_xAlarmActive;

fbKochModuleNotReady(i_xConditions := CFG_MC.Generic.KochModulePresent AND NOT MC_InputOutput.Network.Machine.Commands.KochModuleReady);
MC_InputOutput.Network.Machine.Exceptions.KochModuleNotReady	:= fbKochModuleNotReady.q_xAlarmActive;

IF tofReactionActive.Q  THEN
	xReactionReadyToBePerformed	:=	FALSE;
END_IF

END_STEP
STEP Output:
// Encoder Emulation Management
fbEncoderEmulation(i_xErrorReset :=	VAR_Machine.iq_stCmd.i_xReset, i_xEnable := xEncEmulationEnable);
VAR_Machine.iq_stStatus.q_xEncoderEmulationError	:= fbEncoderEmulation.q_xError;

// Output
tofInMotionTimerDone(IN:= 	VAR_Machine.stMasterModule.iq_stStatus.q_xPhaseShiftDone	OR
							VAR_Machine.stFillerModule.iq_stStatus.q_xPhaseShiftDone	OR
							VAR_Machine.stInletModule.iq_stStatus.q_xPhaseShiftDone		OR
							VAR_Machine.stOutletModule.iq_stStatus.q_xPhaseShiftDone,
							PT := t#1s);

VAR_Machine.iq_stStatus.q_xInMotionTimerDone		:= tofInMotionTimerDone.Q;

MC_InputOutput.Safety.Filler.Status.ModulePowered	:= VAR_Machine.stFillerModule.iq_stStatus.q_xModulePowered;
MC_InputOutput.Safety.Inlet.Status.ModulePowered	:= VAR_Machine.stInletModule.iq_stStatus.q_xModulePowered;
MC_InputOutput.Safety.Outlet.Status.ModulePowered	:= VAR_Machine.stOutletModule.iq_stStatus.q_xModulePowered;

VAR_Machine.iq_stStatus.q_xCombiSynchronized		:= xCombiSynchronized;
VAR_Machine.iq_stStatus.q_xCombiSynchroStopDone		:= xCombiSynchroStopDone;
VAR_Machine.iq_stStatus.q_xCombiFixedSpeed			:= xCombiFixedSpeed;
VAR_Machine.iq_stStatus.q_xCombiSynchroInProgress	:= xCombiSynchroInProgress;

VAR_Machine.iq_stStatus.q_xCombiActive				:= xCombiActive;
VAR_Machine.iq_stStatus.q_xAutoActive				:= xAutoActive	AND
														VAR_Machine.stMasterModule.iq_stStatus.q_xAutoActive	AND
														VAR_Machine.stFillerModule.iq_stStatus.q_xAutoActive	AND
														(VAR_Machine.stOutletModule.iq_stStatus.q_xAutoActive	OR
														NOT VAR_Machine.stOutletModule.iq_stStatus.q_xModuleReal);
VAR_Machine.iq_stStatus.q_xStepByStepActive				:= xStepByStepActive;
VAR_Machine.iq_stStatus.q_xStepByStepSingleAxisActive	:= xStepByStepSingleAxisActive;//V4.A.A.1.7.0
VAR_Machine.iq_stStatus.q_xStepByStepSingAxisRevActive	:= xStepByStepSingleAxisRevActive;//v999
VAR_Machine.iq_stStatus.q_xBrakeReleaseActive			:= xBrakeReleaseActive;
VAR_Machine.iq_stStatus.q_xMultiModalityActive			:= xMultiActive;
VAR_Machine.iq_stStatus.q_xNoModalityactive				:= xNoOpActive;
VAR_Machine.iq_stStatus.q_xPositioningActive			:= xPositioningActive;
VAR_Machine.iq_stStatus.q_xVelocityActive				:= xVelocityActive;
VAR_Machine.iq_stStatus.q_xSelHomingActive				:= xSelHomingActive;
VAR_Machine.iq_stStatus.q_xThirdPartyDynSetupActive		:= xThirdPartySetupActive;
VAR_Machine.iq_stStatus.q_xInductionSetupActive			:= xInductionSetupActive;
VAR_Machine.iq_stStatus.q_xJogActive					:= xJogActive	AND
															VAR_Machine.stMasterModule.iq_stStatus.q_xJogActive		AND
															VAR_Machine.stFillerModule.iq_stStatus.q_xAutoActive	AND
															(VAR_Machine.stOutletModule.iq_stStatus.q_xAutoActive	OR
															NOT VAR_Machine.stOutletModule.iq_stStatus.q_xModuleReal);

IF VAR_Machine.iq_stStatus.q_xMultiModalityActive 			OR
	NOT VAR_Machine.stFillerModule.iq_stStatus.q_xInitDone 	OR
	NOT VAR_Machine.stInletModule.iq_stStatus.q_xInitDone 	OR
	NOT VAR_Machine.stOutletModule.iq_stStatus.q_xInitDone 	THEN

	VAR_Machine.iq_stStatus.q_xMachineStopped		:= TRUE;
ELSE
	VAR_Machine.iq_stStatus.q_xMachineStopped		:= VAR_Machine.stFillerModule.iq_stStatus.q_xModuleStopped		AND
														(VAR_Machine.stInletModule.iq_stStatus.q_xModuleStopped		OR
														NOT VAR_Machine.stInletModule.iq_stStatus.q_xModuleReal)	AND
														(VAR_Machine.stOutletModule.iq_stStatus.q_xModuleStopped	OR
														NOT VAR_Machine.stOutletModule.iq_stStatus.q_xModuleReal);
	VAR_Machine.iq_stStatus.q_xMachineStartFbk		:= (xAutoActive 		AND VAR_Machine.iq_stCmd.i_xStart)			OR
														(xJogActive			AND	VAR_Machine.iq_stCmd.i_xJogPushButton) 	OR
														(xStepByStepActive	AND NOT xStepByStepDone)					OR
														(xStepByStepSingleAxisActive AND NOT xStepByStepSingleAxisDone)  OR
														(xStepByStepSingleAxisRevActive AND NOT xStepByStepSingleAxisReverseDone) OR //v999
														(xPositioningActive AND NOT xPositioningDone)					OR
														(xVelocityActive);
END_IF

VAR_Machine.iq_stStatus.q_xHomed					:= VAR_Machine.stFillerModule.iq_stStatus.q_xModuleHomed	AND
														(VAR_Machine.stOutletModule.iq_stStatus.q_xModuleHomed	OR
														NOT VAR_Machine.stOutletModule.iq_stStatus.q_xModuleReal);
VAR_Machine.iq_stStatus.q_xInPosition				:= xPositioningActive	AND xPositioningDone;
VAR_Machine.iq_stStatus.q_xPowered					:= VAR_Machine.stFillerModule.iq_stStatus.q_xModulePowered		AND
														(VAR_Machine.stOutletModule.iq_stStatus.q_xModulePowered	OR
														NOT VAR_Machine.stOutletModule.iq_stStatus.q_xModuleReal);

VAR_Machine.iq_stStatus.q_xReactionActive			:= tofReactionActive.Q; //xReactionActive;
END_STEP
TRANSITION FROM (Input,SetException,Output) TO Init:=
FALSE
END_TRANSITION
(* @SFCISJUMP := 'Init' *)
END_PROGRAM
```

#### Variables.var - Local variables
```iecst
(*Encoder Emulator*)
VAR
	fbEncoderEmulation : FB_EncEmul;
END_VAR
(*Alarm Core*)
VAR
	xEnableMpAlarmXCore : BOOL;
	fbMpAlarmXCore : MpAlarmXCore;
END_VAR
(* Input Variables *)
VAR
	xInputStepByStepSingleAxisRev : BOOL; (*v999*)
	xInputStepByStepSingleAxis : BOOL; (*//FR*)
	xInputStepByStep : BOOL;
	xInputCombi : BOOL;
	xInputAuto : BOOL;
	xInputVelocity : BOOL;
	xInputSelHoming : BOOL;
	xInputPositioning : BOOL;
	xInputThirdPartySetup : BOOL;
	xInputInductionSetup : BOOL;
	xInputBrakeRelease : BOOL;
	xInputJog : BOOL;
	xInputMulti : BOOL;
	xCombiSynchronized : BOOL;
	xCombiSynchroStopDone : BOOL;
	xCombiFixedSpeed : BOOL;
	xCombiSynchroInProgress : BOOL;
END_VAR
(*Modality Bits*)
VAR
	xAutoMode : BOOL;
	xCombiMode : BOOL;
	xStepByStepSingleAxisReverseMode : BOOL; (*V999*)
	xStepByStepSingleAxisMode : BOOL; (*//FR*)
	xStepByStepMode : BOOL;
	xVelocityMode : BOOL;
	xPositioningMode : BOOL;
	xThirdPartySetupMode : BOOL;
	xInductionSetupMode : BOOL;
	xSelectiveHomingMode : BOOL;
	xBrakeReleaseMode : BOOL;
	xJogMode : BOOL;
	xMultiMode : BOOL;
	xModeReady : BOOL;
	xExitStep : BOOL;
END_VAR
(*Modalities*)
VAR
	xStepByStepSingleAxisReverseDone : BOOL; (*v999*)
	xStepByStepSingleAxisDone : BOOL; (*//FR*)
	xStepByStepDone : BOOL;
	xNoOpActive : BOOL;
	xJogActive : BOOL;
	xMultiActive : BOOL;
	xVelocityActive : BOOL;
	xPositioningDone : BOOL;
	xPositioningActive : BOOL;
	xThirdPartySetupDone : BOOL;
	xThirdPartySetupActive : BOOL;
	xInductionSetupDone : BOOL;
	xInductionSetupActive : BOOL;
	xSelHomingActive : BOOL;
	xStepByStepSingleAxisRevActive : BOOL; (*v999*)
	xStepByStepSingleAxisActive : BOOL; (*//FR*)
	xStepByStepActive : BOOL;
	xBrakeReleaseActive : BOOL;
	xCombiActive : BOOL;
	xAutoActive : BOOL;
END_VAR
(*Steps*)
VAR
	uiStepByStepSingleReverseAxis : UINT; (*v999*)
	uiStepByStepSingleAxis : UINT; (*//FR*)
	uiStepByStep : UINT;
	uiCombiStep : UINT;
	uiAutoStep : UINT;
	uiVelocityStep : UINT;
	uiPositioningStep : UINT;
	uiThirdPartySetupStep : UINT;
	uiInductionSetupStep : UINT;
	uiBrakeReleaseStep : UINT;
	uiSelectiveHomingStep : UINT;
	uiMachinePositioningStep : UINT;
	uiJogStep : UINT;
	uiFillerMultiStep : UINT;
	uiOutletMultiStep : UINT;
	uiInletMultiStep : UINT;
END_VAR
(*Short Int*)
VAR
	uiOldAxisSelected : UINT;
	uiTemp : UINT;
END_VAR
(*Variables*)
VAR
	rOldDecelerationValue : REAL := 100;
	rOldAccelerationValue : REAL := 100;
	xReactionActive : BOOL;
	tofInMotionTimerDone : TOF;
	tofReactionActive : TOF;
	tonClockGeneration : TON; (*v1.7.2*)
	tonFanSeamerActive : TON;
	xEncEmulationEnable : BOOL;
END_VAR
(*Machine Reaction*)
VAR
	fbKochModuleNotReady : FB_ExceptionAlarmX;
	fbQuickStopFromPlc : FB_ExceptionAlarmX;
	fbSeamerFanFault : FB_ExceptionAlarmX;
END_VAR
(*Reaction bits*)
VAR
	xReactionMachineQuickStop : BOOL;
	xReactMasterStop : BOOL;
	xReactMasterQuickStop : BOOL;
	xReactMasterShutdown : BOOL;
	xReactFillerStop : BOOL;
	xReactFillerQuickStop : BOOL;
	xReactFillerEmergencyStop : BOOL;
	xReactInletStop : BOOL;
	xReactInletQuickStop : BOOL;
	xReactInletEmergencyStop : BOOL;
	xReactOutletStop : BOOL;
	xReactOutletQuickStop : BOOL;
	xReactOutletEmergencyStop : BOOL;
	xReactionOnFillerModule : BOOL;
	xReactionOnOutletModule : BOOL;
	xReactionOnInletModule : BOOL;
	xReactionReadyToBePerformed : BOOL;
END_VAR
(*Slow motion command*)
VAR
	xSlowMotionCommandOutlet : BOOL := FALSE;
	xSlowMotionCommandOutletForward : BOOL := FALSE;
	xSlowMotionCommandOutletBackward : BOOL := FALSE;
	xSlowMotionCommandInlet : BOOL := FALSE;
	xSlowMotionCommandInletForward : BOOL := FALSE;
	xSlowMotionCommandInletBackward : BOOL := FALSE;
	uiMinRealFillerIndex : UINT;
	uiMaxRealFillerIndex : UINT;
	uiAxisIndex : UINT;
	uiMaxRealInletIndex : UINT;
	uiMinRealOutletIndex : UINT;
END_VAR
```

### Program Logical/30_MC/Task/Cyclic02/MC_MASTER (IEC) - MC_MASTER - C#1 0.8ms or C#2 10.4ms

#### Cyclic.sfc - Cyclic code
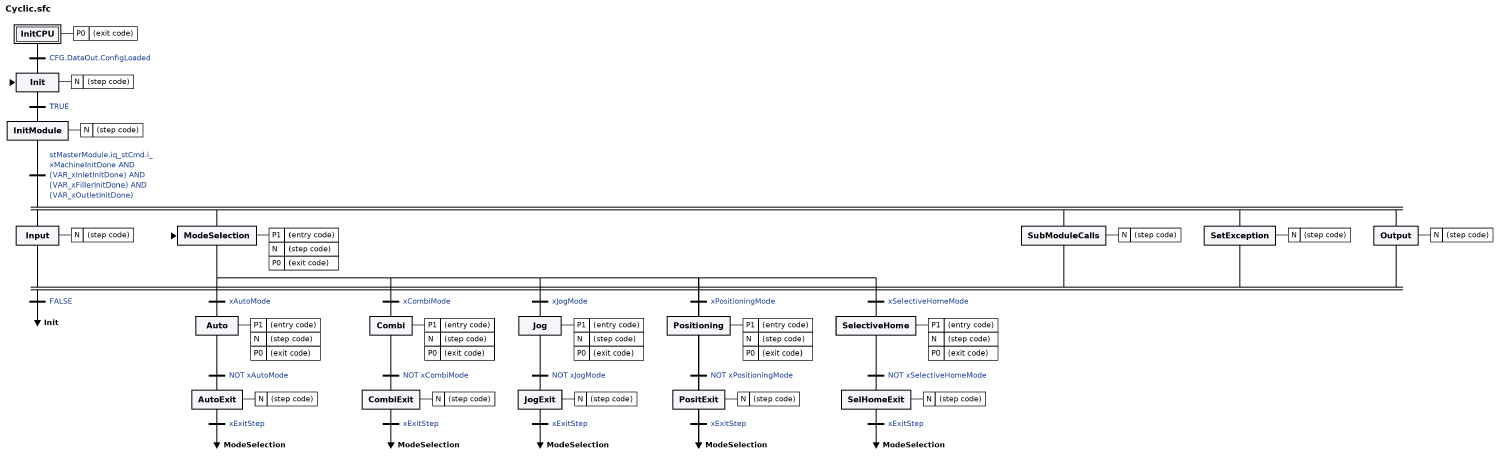
```iecst
PROGRAM _CYCLIC
INITIAL_STEP InitCPU:
END_STEP
EXIT_ACTION
VAR_EmergencyDec := FC_GetAccFromTimeAndJerk(	CFG_MC.Movements.EmergencyDec,
												CFG_MC.Movements.Jerk,
												CFG_MC.Movements.MachineMaxSpeed / 10.0);

VAR_ShutDownDec := FC_GetAccFromTimeAndJerk(	CFG_MC.Movements.ShutDownDec,
												0.0,
												CFG_MC.Movements.MachineMaxSpeed / 10.0);
END_ACTION
TRANSITION FROM InitCPU TO Init:=
CFG.DataOut.ConfigLoaded
END_TRANSITION
STEP Init:
FOR uiAxisIndex := CST_MachineMasterAxis TO CST_NumberOfAxesMasterModule BY 1 DO
	stMasterModule.iq_astSubModuleAxis[uiAxisIndex].iq_stParam.i_rEndlessJerk			:= CFG_MC.Movements.Jerk;
	stMasterModule.iq_astSubModuleAxis[uiAxisIndex].iq_stParam.i_rEmergencyDeceleration	:= VAR_EmergencyDec;
	stMasterModule.iq_astSubModuleAxis[uiAxisIndex].iq_stParam.i_rShutdownDeceleration	:= VAR_ShutDownDec;
	stMasterModule.iq_astSubModuleAxis[uiAxisIndex].iq_stParam.i_rJogDeceleration		:= CST_JogDeceleration;
END_FOR
END_STEP
TRANSITION FROM Init TO InitModule:=
TRUE
END_TRANSITION
STEP InitModule:
(* Alarm initialization *)
fbPwr01Fault.i_psAlarmName					:=	ADR('PowerFault01');
fbPwr01Fault.i_pstMpAlarmXLink				:=	ADR(gMasterAlarmXCoreLink);
fbPwr01Fault.i_pxAcknowledge				:=	ADR(stMasterModule.iq_stCmd.i_xReset);
fbPwr01Fault.i_pxInitCoreDone				:=	ADR(stMasterModule.iq_stCmd.i_xAlarmInitOk);
fbPwr01Fault.i_xAutoAck						:=	FALSE;

fbPwr02Fault.i_psAlarmName					:=	ADR('PowerFault02');
fbPwr02Fault.i_pstMpAlarmXLink				:=	ADR(gMasterAlarmXCoreLink);
fbPwr02Fault.i_pxAcknowledge				:=	ADR(stMasterModule.iq_stCmd.i_xReset);
fbPwr02Fault.i_pxInitCoreDone				:=	ADR(stMasterModule.iq_stCmd.i_xAlarmInitOk);
fbPwr02Fault.i_xAutoAck						:=	FALSE;

fbPwr01Error.i_psAlarmName					:=	ADR('Power01Error');
fbPwr01Error.i_pstMpAlarmXLink				:=	ADR(gMasterAlarmXCoreLink);
fbPwr01Error.i_pxAcknowledge				:=	ADR(stMasterModule.iq_stCmd.i_xReset);
fbPwr01Error.i_pxInitCoreDone				:=	ADR(stMasterModule.iq_stCmd.i_xAlarmInitOk);
fbPwr01Error.i_xAutoAck						:=	FALSE;

fbPwr02Error.i_psAlarmName					:=	ADR('Power02Error');
fbPwr02Error.i_pstMpAlarmXLink				:=	ADR(gMasterAlarmXCoreLink);
fbPwr02Error.i_pxAcknowledge				:=	ADR(stMasterModule.iq_stCmd.i_xReset);
fbPwr02Error.i_pxInitCoreDone				:=	ADR(stMasterModule.iq_stCmd.i_xAlarmInitOk);
fbPwr02Error.i_xAutoAck						:=	FALSE;

fbPwr01BleederFault.i_psAlarmName			:=	ADR('BleederFault01');
fbPwr01BleederFault.i_pstMpAlarmXLink		:=	ADR(gMasterAlarmXCoreLink);
fbPwr01BleederFault.i_pxAcknowledge			:=	ADR(stMasterModule.iq_stCmd.i_xReset);
fbPwr01BleederFault.i_pxInitCoreDone		:=	ADR(stMasterModule.iq_stCmd.i_xAlarmInitOk);
fbPwr01BleederFault.i_xAutoAck				:=	FALSE;

fbPwr02BleederFault.i_psAlarmName			:=	ADR('BleederFault02');
fbPwr02BleederFault.i_pstMpAlarmXLink		:=	ADR(gMasterAlarmXCoreLink);
fbPwr02BleederFault.i_pxAcknowledge			:=	ADR(stMasterModule.iq_stCmd.i_xReset);
fbPwr02BleederFault.i_pxInitCoreDone		:=	ADR(stMasterModule.iq_stCmd.i_xAlarmInitOk);
fbPwr02BleederFault.i_xAutoAck				:=	FALSE;

fbMasterError.i_psAlarmName					:=	ADR('MasterAxisError');
fbMasterError.i_pstMpAlarmXLink				:=	ADR(gMasterAlarmXCoreLink);
fbMasterError.i_pxAcknowledge				:=	ADR(stMasterModule.iq_stCmd.i_xReset);
fbMasterError.i_pxInitCoreDone				:=	ADR(stMasterModule.iq_stCmd.i_xAlarmInitOk);
fbMasterError.i_xAutoAck					:=	FALSE;

(******************** Axes function block initialization **************************)
(* POWER SUPPLY 1 *)
fbPowerSupply01.i_xEnable						:=	TRUE;
fbPowerSupply01.i_xToken						:=	TRUE;
fbPowerSupply01.i_pAxisADR 						:=	ADR(VAR_AxPowerSupply01);
fbPowerSupply01.i_pAxisMpLink					:=	ADR(gMasterPwr01Link);
fbPowerSupply01.i_pSecondaryAxisADR				:=	0;
fbPowerSupply01.i_pSecondaryAxisMpLink			:=	0;
fbPowerSupply01.i_pstCmd						:=	ADR(stMasterModule.iq_astSubModuleAxis[CST_MasterPowerSupply01].iq_stCmd);
fbPowerSupply01.i_pstParameter					:=	ADR(stMasterModule.iq_astSubModuleAxis[CST_MasterPowerSupply01].iq_stParam);
fbPowerSupply01.i_pstStatus						:=	ADR(stMasterModule.iq_astSubModuleAxis[CST_MasterPowerSupply01].iq_stStatus);
fbPowerSupply01.i_pstAxisHome					:=	ADR(VAR_PowerSupplyHomeData);

stMasterModule.iq_astSubModuleAxis[CST_MasterPowerSupply01].iq_stParam.i_xMachineMaster		:=	FALSE;
stMasterModule.iq_astSubModuleAxis[CST_MasterPowerSupply01].iq_stParam.i_udiMasterLink		:=	ADR(gMasterPwr01Link);

(* POWER SUPPLY 2 *)
fbPowerSupply02.i_xEnable						:=	TRUE;
fbPowerSupply02.i_xToken						:=	TRUE;
fbPowerSupply02.i_pAxisADR 						:=	ADR(VAR_AxPowerSupply02);
fbPowerSupply02.i_pAxisMpLink					:=	ADR(gMasterPwr02Link);
fbPowerSupply02.i_pSecondaryAxisADR				:=	0;
fbPowerSupply02.i_pSecondaryAxisMpLink			:=	0;
fbPowerSupply02.i_pstCmd						:=	ADR(stMasterModule.iq_astSubModuleAxis[CST_MasterPowerSupply02].iq_stCmd);
fbPowerSupply02.i_pstParameter					:=	ADR(stMasterModule.iq_astSubModuleAxis[CST_MasterPowerSupply02].iq_stParam);
fbPowerSupply02.i_pstStatus						:=	ADR(stMasterModule.iq_astSubModuleAxis[CST_MasterPowerSupply02].iq_stStatus);
fbPowerSupply02.i_pstAxisHome					:=	ADR(VAR_PowerSupplyHomeData);

stMasterModule.iq_astSubModuleAxis[CST_MasterPowerSupply02].iq_stParam.i_xMachineMaster		:=	FALSE;
stMasterModule.iq_astSubModuleAxis[CST_MasterPowerSupply02].iq_stParam.i_udiMasterLink		:=	ADR(gMasterPwr02Link);

(* MACHINE MASTER AXIS *)
fbMachineMasterSlow.i_xEnable 					:= TRUE;	//v1.66
fbMachineMasterSlow.i_xToken					:= TRUE;	//v1.66
fbMachineMasterSlow.i_xVelocityControl 			:= FALSE;	//v1.66
fbMachineMasterSlow.i_xThirdPartyMotor			:= FALSE;	//v1.66
fbMachineMasterSlow.i_pAxisMpLink				:= ADR(gMasterLink);	//v1.66
fbMachineMasterSlow.i_pAxisADR					:= ADR(VAR_AxMachineMaster);	//v1.66
fbMachineMasterSlow.i_pSecondaryAxisMpLink		:= 0;	//v1.66
fbMachineMasterSlow.i_pSecondaryAxisADR			:= 0;	//v1.66

fbMachineMasterSlow.i_pstCmd					:= ADR(stMasterModule.iq_astSubModuleAxis[CST_MachineMasterAxis].iq_stCmd);	//v1.66
fbMachineMasterSlow.i_pstParameter				:= ADR(stMasterModule.iq_astSubModuleAxis[CST_MachineMasterAxis].iq_stParam);	//v1.66
fbMachineMasterSlow.i_pstStatus					:= ADR(stMasterModule.iq_astSubModuleAxis[CST_MachineMasterAxis].iq_stStatus);	//v1.66
fbMachineMasterSlow.i_pstAxisHome				:= ADR(VAR_AxMachineMasterHomeData);	//v1.66

stMasterModule.iq_astSubModuleAxis[CST_MachineMasterAxis].iq_stParam.i_xMachineMaster		:= TRUE;
stMasterModule.iq_astSubModuleAxis[CST_MachineMasterAxis].iq_stParam.i_udiMasterLink		:= ADR(gMasterLink);
stMasterModule.iq_astSubModuleAxis[CST_MachineMasterAxis].iq_stParam.i_udiHomingPosition	:= ADR(stMasterModule.iq_stParameters.i_lrRephasingPosition);
//V4.A.A.1.6.10a
IF stMasterModule.iq_astSubModuleAxis[CST_MachineMasterAxis].iq_stParam.i_prMasterVelocity	=0 THEN
	stMasterModule.iq_astSubModuleAxis[CST_MachineMasterAxis].iq_stParam.i_prMasterVelocity	:= ADR(stMasterModule.iq_astSubModuleAxis[CST_MachineMasterAxis].iq_stStatus.q_stMainAxisStatus.q_rVelocity);
END_IF

//Master Virtual Axis - HMI Presence
HMI_MC_AxisPresent._99 := TRUE;
//NEW MANAGEMENT //FR
HMI_MC_GenericAxisDataNew[1].xHmiPresent 	:= TRUE;
HMI_MC_GenericAxisDataNew[1].uiAxisID		:= 99;
HMI_MC_GenericAxisDataNew[1].usiHmiName		:= 99;
END_STEP
TRANSITION Machine init done FROM InitModule TO (Input,ModeSelection,SubModuleCalls,SetException,Output):=
stMasterModule.iq_stCmd.i_xMachineInitDone AND
(VAR_xInletInitDone) AND
(VAR_xFillerInitDone) AND
(VAR_xOutletInitDone)  //v4.A.A.1.6.7
END_TRANSITION
STEP Input:
(* Reset Command To All Axes *)
FOR uiAxisIndex := CST_MachineMasterAxis TO CST_NumberOfAxesMasterModule BY 1 DO
	stMasterModule.iq_astSubModuleAxis[uiAxisIndex].iq_stParam.i_rStopPosition	:=	stMasterModule.iq_stParameters.i_rStopPosition;

	stMasterModule.iq_astSubModuleAxis[uiAxisIndex].iq_stCmd.i_xErrorReset				:=	stMasterModule.iq_stCmd.i_xReset;
	stMasterModule.iq_astSubModuleAxis[uiAxisIndex].iq_stParam.i_rEndlessAcceleration	:=	stMasterModule.iq_stParameters.i_rEndlessAcceleration;
	stMasterModule.iq_astSubModuleAxis[uiAxisIndex].iq_stParam.i_rEndlessDeceleration	:=	stMasterModule.iq_stParameters.i_rEndlessDeceleration;
END_FOR

(******* Spread the reaction to the axes ********)
(* Quick stop *)
stMasterModule.iq_astSubModuleAxis[CST_MachineMasterAxis].iq_stCmd.i_xQuickStop		:= stMasterModule.iq_stCmd.i_xQuickStop;
(* Emergency stop *)
stMasterModule.iq_astSubModuleAxis[CST_MachineMasterAxis].iq_stCmd.i_xEmergencyStop	:= stMasterModule.iq_stCmd.i_xEmergencyStop OR (NOT stMasterModule.iq_stCmd.i_xJogPB AND stMasterModule.iq_stCmd.i_xJogMode AND NOT stMasterModule.iq_astSubModuleAxis[CST_MachineMasterAxis].iq_stStatus.q_stMainAxisStatus.q_xStopped);
(* Shutdown *)
stMasterModule.iq_astSubModuleAxis[CST_MachineMasterAxis].iq_stCmd.i_xShutdown		:= stMasterModule.iq_stCmd.i_xShutdown;

xReactionActive := stMasterModule.iq_stCmd.i_xQuickStop OR stMasterModule.iq_stCmd.i_xEmergencyStop OR stMasterModule.iq_stCmd.i_xShutdown OR (NOT stMasterModule.iq_stCmd.i_xJogPB AND stMasterModule.iq_stCmd.i_xJogMode AND NOT stMasterModule.iq_astSubModuleAxis[CST_MachineMasterAxis].iq_stStatus.q_stMainAxisStatus.q_xStopped);

tofReactionActive(IN := xReactionActive, PT := t#100ms);

(* Input Signals *)
xInputAuto			:= stMasterModule.iq_stCmd.i_xAutoMode;
xInputJog			:= stMasterModule.iq_stCmd.i_xJogMode;
xInputCombi			:= stMasterModule.iq_stCmd.i_xCombi;
xInputPositioning	:= stMasterModule.iq_stCmd.i_xPositioning;
xInputSelHoming		:= stMasterModule.iq_stCmd.i_xSelectiveHomingMode;

fbMachineMasterFast.i_xCmdEnableCurves	:= stMasterModule.iq_stCmd.i_xEnableCurves;	//V4.A.A.1.6.10
END_STEP
STEP ModeSelection:
xNoOpActive			:= TRUE;
xAutoActive 		:= FALSE;
xPositioningActive 	:= FALSE;
xJogActive			:= FALSE;
xCombiActive 		:= FALSE;
xPositioningActive	:= FALSE;

// Change status
xModeReady	:=	NOT xAutoMode 			AND
				NOT xCombiMode			AND
				NOT xJogMode 			AND
				NOT xPositioningMode	AND
				NOT tofReactionActive.Q;

IF xModeReady THEN
	IF xInputAuto THEN
		xAutoMode := TRUE;
	ELSIF xInputPositioning THEN
		xPositioningMode := TRUE;
	ELSIF xInputJog THEN
		xJogMode := TRUE;
	ELSIF xInputCombi THEN
		xCombiMode := TRUE;
	ELSIF xInputSelHoming THEN
		xSelectiveHomeMode := TRUE;
	END_IF
END_IF
END_STEP
ENTRY_ACTION
xExitStep		:= FALSE;
stMasterModule.iq_stStatus.q_xMasterRephased	:= FALSE;
END_ACTION
EXIT_ACTION
xNoOpActive := FALSE;
END_ACTION
TRANSITION FROM ModeSelection TO Auto:=
xAutoMode
END_TRANSITION
TRANSITION FROM ModeSelection TO Combi:=
xCombiMode
END_TRANSITION
STEP Combi:
IF xReactionActive OR NOT xInputCombi THEN
	xCombiMode	:=	FALSE;
END_IF

CASE uiCombiStep OF
	0:
		IF stMasterModule.iq_astSubModuleAxis[CST_MachineMasterAxis].iq_stStatus.q_stMainAxisStatus.q_xReadyForACommand	THEN
			IF 	stMasterModule.iq_astSubModuleAxis[CST_MachineMasterAxis].iq_stStatus.q_stMainAxisStatus.q_xSynchroWithOffset THEN
				stMasterModule.iq_astSubModuleAxis[CST_MachineMasterAxis].iq_stCmd.i_xPhaseCompensation	:=	TRUE;
				uiCombiStep	:= 50;
			ELSE
				uiCombiStep	:= 100;
			END_IF
		END_IF

	50:
		IF NOT stMasterModule.iq_astSubModuleAxis[CST_MachineMasterAxis].iq_stStatus.q_stMainAxisStatus.q_xSynchroWithOffset THEN
			stMasterModule.iq_astSubModuleAxis[CST_MachineMasterAxis].iq_stCmd.i_xPhaseCompensation	:=	FALSE;
			uiCombiStep	:= 100;
		END_IF

	100:
		IF stMasterModule.iq_stCmd.i_xMasterRephasingRequest THEN
			stMasterModule.iq_astSubModuleAxis[CST_MachineMasterAxis].iq_stCmd.i_xHome	:= TRUE;
			IF NOT stMasterModule.iq_astSubModuleAxis[CST_MachineMasterAxis].iq_stStatus.q_stMainAxisStatus.q_xIsHomed THEN
				uiCombiStep	:= 110;
			END_IF
		ELSE
			uiCombiStep	:= 130;
		END_IF

	110:
		IF stMasterModule.iq_astSubModuleAxis[CST_MachineMasterAxis].iq_stStatus.q_stMainAxisStatus.q_xIsHomed THEN
			stMasterModule.iq_astSubModuleAxis[CST_MachineMasterAxis].iq_stCmd.i_xHome	:= FALSE;
			uiCombiStep	:= 120;
		END_IF

	120:
		stMasterModule.iq_stStatus.q_xMasterRephased	:= TRUE;
		uiCombiStep										:= 130;

	130:
		stMasterModule.iq_astSubModuleAxis[CST_MachineMasterAxis].iq_stCmd.i_xGear	:= stMasterModule.iq_stCmd.i_xStart;
		uiCombiStep	:=	140;

	140:(* Wait the synchro stop command or not start command *)
		IF NOT stMasterModule.iq_stCmd.i_xStart OR stMasterModule.iq_stCmd.i_xCombiSynchroStop THEN
			stMasterModule.iq_astSubModuleAxis[CST_MachineMasterAxis].iq_stCmd.i_xGear := FALSE;
			IF stMasterModule.iq_astSubModuleAxis[CST_MachineMasterAxis].iq_stStatus.q_stMainAxisStatus.q_xStopped OR NOT stMasterModule.iq_stCmd.i_xStart THEN
				xCombiSynchroStopDone := TRUE;
				uiCombiStep	:= 180;
			ELSE
				stMasterModule.iq_astSubModuleAxis[CST_MachineMasterAxis].iq_stCmd.i_xMoveVelocity		:= TRUE;
				stMasterModule.iq_astSubModuleAxis[CST_MachineMasterAxis].iq_stParam.i_rEndlessVelocity	:= stMasterModule.iq_astSubModuleAxis[CST_MachineMasterAxis].iq_stStatus.q_stMainAxisStatus.q_rVelocity;
				uiCombiStep	:=	150;
			END_IF
		ELSIF stMasterModule.iq_stCmd.i_xPhaseShift	THEN (* One pitch command *)
			stMasterModule.iq_astSubModuleAxis[CST_MachineMasterAxis].iq_stParam.i_rPhaseShiftDistance	:= stMasterModule.iq_stParameters.i_rPhaseShiftDistance;
			stMasterModule.iq_astSubModuleAxis[CST_MachineMasterAxis].iq_stCmd.i_xPhaseShift	:= TRUE;
			uiCombiStep	:=	400;
		ELSIF stMasterModule.iq_stCmd.i_xOnePitchShift THEN
			stMasterModule.iq_astSubModuleAxis[CST_MachineMasterAxis].iq_stCmd.i_xOnePitchShift	:= TRUE;
			uiCombiStep	:=	300;
		END_IF

	150:(* Combi synchro stop in progress *)
		xCombiSynchroStopDone	:= TRUE;
		IF NOT stMasterModule.iq_stCmd.i_xStart THEN
			stMasterModule.iq_astSubModuleAxis[CST_MachineMasterAxis].iq_stCmd.i_xMoveVelocity	:= FALSE;
			uiCombiStep	:=	180;
		END_IF

	180:(* Combi synchro stop in progress *)
		IF stMasterModule.iq_astSubModuleAxis[CST_MachineMasterAxis].iq_stStatus.q_stMainAxisStatus.q_xStopped THEN
			xCombiSynchroStopDone	:= FALSE;
			IF stMasterModule.iq_astSubModuleAxis[CST_MachineMasterAxis].iq_stStatus.q_stMainAxisStatus.q_xSynchroWithOffset	AND
				stMasterModule.iq_astSubModuleAxis[CST_MachineMasterAxis].iq_stStatus.q_stMainAxisStatus.q_xReadyForACommand	THEN

				stMasterModule.iq_astSubModuleAxis[CST_MachineMasterAxis].iq_stCmd.i_xPhaseCompensation	:=	TRUE;
				uiCombiStep	:=	200;
			END_IF
		END_IF

		IF stMasterModule.iq_astSubModuleAxis[CST_MachineMasterAxis].iq_stStatus.q_stMainAxisStatus.q_xStopped AND
			stMasterModule.iq_stCmd.i_xStart					AND
			NOT stMasterModule.iq_stCmd.i_xCombiSynchroStop		THEN

			uiCombiStep	:=	130;
		END_IF

	200:
		IF NOT stMasterModule.iq_astSubModuleAxis[CST_MachineMasterAxis].iq_stStatus.q_stMainAxisStatus.q_xSynchroWithOffset THEN
			stMasterModule.iq_astSubModuleAxis[CST_MachineMasterAxis].iq_stCmd.i_xPhaseCompensation	:= FALSE;
			uiCombiStep	:=	180;
		END_IF

	300:
		stMasterModule.iq_stStatus.q_xOnePitchShifDone	:= stMasterModule.iq_astSubModuleAxis[CST_MachineMasterAxis].iq_stStatus.q_stMainAxisStatus.q_xOnePitchShiftDone;

		(* Synchro stop command *)
		IF NOT stMasterModule.iq_stCmd.i_xStart OR stMasterModule.iq_stCmd.i_xCombiSynchroStop OR
			stMasterModule.iq_astSubModuleAxis[CST_MachineMasterAxis].iq_stStatus.q_stMainAxisStatus.q_xOnePitchShiftDone AND NOT
			stMasterModule.iq_stCmd.i_xOnePitchShift THEN

			stMasterModule.iq_astSubModuleAxis[CST_MachineMasterAxis].iq_stCmd.i_xOnePitchShift	:= FALSE;
			stMasterModule.iq_stStatus.q_xOnePitchShifDone	:= FALSE;

			uiCombiStep	:= 140;
		END_IF

	400:
		stMasterModule.iq_stStatus.q_xPhaseShiftDone	:= stMasterModule.iq_astSubModuleAxis[CST_MachineMasterAxis].iq_stStatus.q_stMainAxisStatus.q_xPhaseShiftDone;
		(* Synchro stop command *)
		IF NOT stMasterModule.iq_stCmd.i_xStart OR stMasterModule.iq_stCmd.i_xCombiSynchroStop OR
			stMasterModule.iq_astSubModuleAxis[CST_MachineMasterAxis].iq_stStatus.q_stMainAxisStatus.q_xPhaseShiftDone AND NOT
			stMasterModule.iq_stCmd.i_xPhaseShift THEN

			stMasterModule.iq_astSubModuleAxis[CST_MachineMasterAxis].iq_stCmd.i_xPhaseShift := FALSE;
			stMasterModule.iq_stStatus.q_xPhaseShiftDone := FALSE;
			uiCombiStep	:= 140;
		END_IF
END_CASE
END_STEP
ENTRY_ACTION
uiCombiStep	 			:= 0;
xCombiActive 			:= TRUE;
xCombiSynchroStopDone	:= FALSE;
END_ACTION
EXIT_ACTION
stMasterModule.iq_astSubModuleAxis[CST_MachineMasterAxis].iq_stCmd.i_xHome			:= FALSE;
stMasterModule.iq_astSubModuleAxis[CST_MachineMasterAxis].iq_stCmd.i_xMoveVelocity	:= FALSE;
stMasterModule.iq_astSubModuleAxis[CST_MachineMasterAxis].iq_stCmd.i_xGear			:= FALSE;
stMasterModule.iq_astSubModuleAxis[CST_MachineMasterAxis].iq_stCmd.i_xOnePitchShift	:= FALSE;
stMasterModule.iq_astSubModuleAxis[CST_MachineMasterAxis].iq_stCmd.i_xPhaseCompensation	:= FALSE;

stMasterModule.iq_stStatus.q_xOnePitchShifDone	:= FALSE;
END_ACTION
TRANSITION FROM Combi TO CombiExit:=
NOT xCombiMode
END_TRANSITION
STEP CombiExit:
stMasterModule.iq_astSubModuleAxis[CST_MachineMasterAxis].iq_stCmd.i_xGear := FALSE;
xCombiSynchroStopDone	:= FALSE;

IF stMasterModule.iq_stStatus.q_xModuleStopped THEN
	xExitStep	:=	TRUE;
END_IF
END_STEP
TRANSITION FROM CombiExit TO ModeSelection:=
xExitStep
END_TRANSITION
(* @SFCISJUMP := 'ModeSelection' *)
TRANSITION FROM ModeSelection TO Jog:=
xJogMode
END_TRANSITION
STEP Jog:
IF xReactionActive OR NOT xInputJog THEN
	xJogMode	:= FALSE;
END_IF

xJogActive	:= TRUE;

CASE uiJogStep OF
	0:
		IF stMasterModule.iq_astSubModuleAxis[CST_MachineMasterAxis].iq_stStatus.q_stMainAxisStatus.q_xReadyForACommand THEN
			IF stMasterModule.iq_astSubModuleAxis[CST_MachineMasterAxis].iq_stStatus.q_stMainAxisStatus.q_xSynchroWithOffset THEN
				stMasterModule.iq_astSubModuleAxis[CST_MachineMasterAxis].iq_stCmd.i_xPhaseCompensation	:= TRUE;
				uiJogStep	:= 50;
			ELSE
				uiJogStep	:= 100;
			END_IF
		END_IF

	50:
		IF NOT stMasterModule.iq_astSubModuleAxis[CST_MachineMasterAxis].iq_stStatus.q_stMainAxisStatus.q_xSynchroWithOffset THEN
			stMasterModule.iq_astSubModuleAxis[CST_MachineMasterAxis].iq_stCmd.i_xPhaseCompensation	:= FALSE;
			uiJogStep	:= 100;
		END_IF

	100:
		IF stMasterModule.iq_stCmd.i_xMasterRephasingRequest THEN
			stMasterModule.iq_astSubModuleAxis[CST_MachineMasterAxis].iq_stCmd.i_xHome	:= TRUE;
			uiJogStep	:= 110;
		ELSE
			uiJogStep	:= 130;
		END_IF

	110:
		IF stMasterModule.iq_astSubModuleAxis[CST_MachineMasterAxis].iq_stStatus.q_stMainAxisStatus.q_xIsHomed	THEN
			stMasterModule.iq_astSubModuleAxis[CST_MachineMasterAxis].iq_stCmd.i_xHome	:= FALSE;
			uiJogStep	:= 120;
		END_IF

	120:
		stMasterModule.iq_stStatus.q_xMasterRephased	:= TRUE;
		uiJogStep										:= 130;

	130:
		stMasterModule.iq_astSubModuleAxis[CST_MachineMasterAxis].iq_stParam.i_rJogVelocity	:= MAX(1, stMasterModule.iq_stParameters.i_rJogVelocity);
		stMasterModule.iq_astSubModuleAxis[CST_MachineMasterAxis].iq_stCmd.i_xJogPositive	:= stMasterModule.iq_stCmd.i_xJogPB;
END_CASE
END_STEP
ENTRY_ACTION
uiJogStep	:= 0;
xJogActive	:= TRUE;
END_ACTION
EXIT_ACTION
stMasterModule.iq_astSubModuleAxis[CST_MachineMasterAxis].iq_stCmd.i_xHome	:= FALSE;
END_ACTION
TRANSITION FROM Jog TO JogExit:=
NOT xJogMode
END_TRANSITION
STEP JogExit:
stMasterModule.iq_astSubModuleAxis[CST_MachineMasterAxis].iq_stCmd.i_xJogPositive := FALSE;

IF stMasterModule.iq_stStatus.q_xModuleStopped THEN
	xExitStep	:= TRUE;
END_IF
END_STEP
TRANSITION FROM JogExit TO ModeSelection:=
xExitStep
END_TRANSITION
(* @SFCISJUMP := 'ModeSelection' *)
TRANSITION FROM ModeSelection TO Positioning:=
xPositioningMode
END_TRANSITION
STEP Positioning:
IF xReactionActive OR NOT xInputPositioning THEN
	xPositioningMode	:= FALSE;
END_IF

xPositioningActive	:= TRUE;

CASE uiPositioningStep OF
	0:
		IF stMasterModule.iq_astSubModuleAxis[CST_MachineMasterAxis].iq_stStatus.q_stMainAxisStatus.q_xReadyForACommand	THEN
			uiPositioningStep	:= 100;
		END_IF

	100:
		IF stMasterModule.iq_stCmd.i_xMasterRephasingRequest THEN
			stMasterModule.iq_astSubModuleAxis[CST_MachineMasterAxis].iq_stCmd.i_xHome	:= TRUE;
			IF NOT stMasterModule.iq_astSubModuleAxis[CST_MachineMasterAxis].iq_stStatus.q_stMainAxisStatus.q_xIsHomed THEN
				uiPositioningStep	:= 110;
			END_IF
		ELSE
			uiPositioningStep	:= 130;
		END_IF

	110:
		IF stMasterModule.iq_astSubModuleAxis[CST_MachineMasterAxis].iq_stStatus.q_stMainAxisStatus.q_xIsHomed THEN
			stMasterModule.iq_astSubModuleAxis[CST_MachineMasterAxis].iq_stCmd.i_xHome	:= FALSE;
			uiPositioningStep	:= 120;
		END_IF

	120:
		stMasterModule.iq_stStatus.q_xMasterRephased	:= TRUE;
		uiPositioningStep								:= 130;

	130:
		IF stMasterModule.iq_stCmd.i_xStart THEN
			rAxisDistance		:= stMasterModule.iq_stParameters.i_rPositioningOffset;
			uiPositioningStep	:= 140;
		END_IF

	140:
		IF stMasterModule.iq_stCmd.i_xStart THEN
			stMasterModule.iq_astSubModuleAxis[CST_MachineMasterAxis].iq_stParam.i_lrAdditiveDistance		:= rAxisDistance;
			stMasterModule.iq_astSubModuleAxis[CST_MachineMasterAxis].iq_stParam.i_rPositioningVelocity		:= 10 * CST_PositioningVel;
			stMasterModule.iq_astSubModuleAxis[CST_MachineMasterAxis].iq_stParam.i_rPositioningAccDec		:= 3 * CST_PositioningAccDec;
			stMasterModule.iq_astSubModuleAxis[CST_MachineMasterAxis].iq_stCmd.i_xMoveAdditive				:= TRUE;
			uiPositioningStep	:=	150;
		END_IF

	150:
		IF NOT stMasterModule.iq_stStatus.q_xModuleStopped THEN
			uiPositioningStep	:= 160;
		END_IF

	160:
		IF stMasterModule.iq_stStatus.q_xModuleStopped AND stMasterModule.iq_astSubModuleAxis[CST_MachineMasterAxis].iq_stStatus.q_stMainAxisStatus.q_xInPosition THEN
			stMasterModule.iq_astSubModuleAxis[CST_MachineMasterAxis].iq_stCmd.i_xMoveAdditive := FALSE;
			uiPositioningStep	:= 170;	//v1.2
		END_IF

	170:	//v1.2
		stMasterModule.iq_stStatus.q_xPositioningDone	:=	TRUE;	//v1.2
END_CASE

END_STEP
ENTRY_ACTION
uiPositioningStep	:= 0;
END_ACTION
EXIT_ACTION
stMasterModule.iq_astSubModuleAxis[CST_MachineMasterAxis].iq_stCmd.i_xHome			:= FALSE;
stMasterModule.iq_astSubModuleAxis[CST_MachineMasterAxis].iq_stCmd.i_xMoveAdditive	:= FALSE;
stMasterModule.iq_stStatus.q_xPositioningDone										:= FALSE;
END_ACTION
TRANSITION FROM Positioning TO PositExit:=
NOT xPositioningMode
END_TRANSITION
STEP PositExit:
IF stMasterModule.iq_stStatus.q_xModuleStopped AND NOT stMasterModule.iq_stCmd.i_xStart THEN
	xExitStep	:= TRUE;
END_IF
END_STEP
TRANSITION FROM PositExit TO ModeSelection:=
xExitStep
END_TRANSITION
(* @SFCISJUMP := 'ModeSelection' *)
TRANSITION FROM ModeSelection TO SelectiveHome:=
xSelectiveHomeMode
END_TRANSITION
STEP SelectiveHome:
xSelHomingActive	:= TRUE;

IF xReactionActive OR NOT xInputSelHoming THEN
	xSelectiveHomeMode	:= FALSE;
END_IF

CASE uiSelectiveHomeStep OF
	0:
		IF stMasterModule.iq_astSubModuleAxis[CST_MachineMasterAxis].iq_stStatus.q_stMainAxisStatus.q_xReadyForACommand	THEN
			uiSelectiveHomeStep	:=	100;
		END_IF

	100:(* If the cyclic communication is on *)
		IF fbMachineMasterFast.q_xCyclicComValid THEN
			fbMachineMasterFast.i_xCmdHoming	:= TRUE;
			uiSelectiveHomeStep	:=	110;
		END_IF

	110:
		IF fbMachineMasterFast.q_xPositionValid AND VAR_AbsEncPerm.xCalibrationDone THEN
			fbMachineMasterFast.i_xCmdHoming	:= FALSE;
			uiSelectiveHomeStep := 120;
		END_IF

	120:
		stMasterModule.iq_stStatus.q_xSelHomingDone	:= TRUE;

END_CASE
END_STEP
ENTRY_ACTION
uiSelectiveHomeStep := 0;
END_ACTION
EXIT_ACTION
stMasterModule.iq_stStatus.q_xSelHomingDone	:=	FALSE;
END_ACTION
TRANSITION FROM SelectiveHome TO SelHomeExit:=
NOT xSelectiveHomeMode
END_TRANSITION
STEP SelHomeExit:
fbMachineMasterFast.i_xCmdHoming	:= FALSE;

xExitStep	:= TRUE;
END_STEP
TRANSITION FROM SelHomeExit TO ModeSelection:=
xExitStep
END_TRANSITION
(* @SFCISJUMP := 'ModeSelection' *)
STEP Auto:
IF xReactionActive OR NOT xInputAuto THEN
	xAutoMode	:=	FALSE;
END_IF

stMasterModule.iq_astSubModuleAxis[CST_MachineMasterAxis].iq_stParam.i_rEndlessVelocity := MAX(1, stMasterModule.iq_stParameters.i_rEndlessVelocity);

CASE uiAutoStep	OF
	0:
		IF stMasterModule.iq_astSubModuleAxis[CST_MachineMasterAxis].iq_stStatus.q_stMainAxisStatus.q_xReadyForACommand THEN
			IF stMasterModule.iq_astSubModuleAxis[CST_MachineMasterAxis].iq_stStatus.q_stMainAxisStatus.q_xSynchroWithOffset THEN
				stMasterModule.iq_astSubModuleAxis[CST_MachineMasterAxis].iq_stCmd.i_xPhaseCompensation	:= TRUE;
				uiAutoStep	:= 50;
			ELSE
				uiAutoStep	:= 100;
			END_IF
		END_IF

	50:
		IF NOT stMasterModule.iq_astSubModuleAxis[CST_MachineMasterAxis].iq_stStatus.q_stMainAxisStatus.q_xSynchroWithOffset THEN
			stMasterModule.iq_astSubModuleAxis[CST_MachineMasterAxis].iq_stCmd.i_xPhaseCompensation	:= FALSE;
			uiAutoStep	:= 100;
		END_IF

	100:
		IF stMasterModule.iq_stCmd.i_xMasterRephasingRequest THEN
			stMasterModule.iq_astSubModuleAxis[CST_MachineMasterAxis].iq_stCmd.i_xHome := TRUE;
			IF NOT stMasterModule.iq_astSubModuleAxis[CST_MachineMasterAxis].iq_stStatus.q_stMainAxisStatus.q_xIsHomed THEN
				uiAutoStep	:= 110;
			END_IF
		ELSE
			uiAutoStep	:= 130;
		END_IF

	110:
		IF stMasterModule.iq_astSubModuleAxis[CST_MachineMasterAxis].iq_stStatus.q_stMainAxisStatus.q_xIsHomed THEN
			stMasterModule.iq_astSubModuleAxis[CST_MachineMasterAxis].iq_stCmd.i_xHome	:= FALSE;
			uiAutoStep	:= 120;
		END_IF

	120:
		stMasterModule.iq_stStatus.q_xMasterRephased	:= TRUE;
		uiAutoStep										:= 130;

	130:
		stMasterModule.iq_astSubModuleAxis[CST_MachineMasterAxis].iq_stCmd.i_xMoveVelocity	:= stMasterModule.iq_stCmd.i_xStart;
END_CASE
END_STEP
ENTRY_ACTION
uiAutoStep	:=	0;
xAutoActive	:=	TRUE;
END_ACTION
EXIT_ACTION
stMasterModule.iq_astSubModuleAxis[CST_MachineMasterAxis].iq_stCmd.i_xHome			:= FALSE;
stMasterModule.iq_astSubModuleAxis[CST_MachineMasterAxis].iq_stCmd.i_xMoveVelocity	:= FALSE;
END_ACTION
TRANSITION FROM Auto TO AutoExit:=
NOT xAutoMode
END_TRANSITION
STEP AutoExit:
stMasterModule.iq_astSubModuleAxis[CST_MachineMasterAxis].iq_stCmd.i_xMoveVelocity := FALSE;

IF stMasterModule.iq_stStatus.q_xModuleStopped THEN
	xExitStep	:= TRUE;
END_IF
END_STEP
TRANSITION FROM AutoExit TO ModeSelection:=
xExitStep
END_TRANSITION
(* @SFCISJUMP := 'ModeSelection' *)
STEP SubModuleCalls:
CASE uiAxisToken OF
	CST_MasterPowerSupply01:
		IF xPowerSupply02 THEN
			uiAxisToken	:= CST_MasterPowerSupply02;
		END_IF

	CST_MasterPowerSupply02:
		uiAxisToken	:=	CST_MasterPowerSupply01;
	ELSE
		uiAxisToken	:=	CST_MasterPowerSupply01;
END_CASE

IF xPowerSupply01 THEN
	fbPowerSupply01.i_xToken	:= uiAxisToken = CST_MasterPowerSupply01;
	fbPowerSupply01;
END_IF

IF xPowerSupply02 THEN
	fbPowerSupply02.i_xToken	:= uiAxisToken = CST_MasterPowerSupply02;
	fbPowerSupply02;
END_IF

stMasterModule.iq_astSubModuleAxis[CST_MachineMasterAxis].iq_stCmd.i_xShutdown	:=
	stMasterModule.iq_astSubModuleAxis[CST_MachineMasterAxis].iq_stCmd.i_xShutdown								OR
	((stMasterModule.iq_astSubModuleAxis[CST_MasterPowerSupply01].iq_stStatus.q_stMainAxisStatus.q_xPowerFault	OR
	stMasterModule.iq_astSubModuleAxis[CST_MasterPowerSupply02].iq_stStatus.q_stMainAxisStatus.q_xPowerFault)	AND CFG_MC.Generic.DisengageImmediately);

fbMachineMasterSlow;
END_STEP
STEP SetException:
(* Set Exception Action *)
fbMpAlarmXCore(MpLink := ADR(gMasterAlarmXCoreLink), Enable := TRUE);
stMasterModule.iq_stStatus.q_xAlarmXCoreEnabled	:= fbMpAlarmXCore.Active;

(* Power fault alarms *)
fbPwr01Fault(i_xConditions := stMasterModule.iq_astSubModuleAxis[CST_MasterPowerSupply01].iq_stStatus.q_stMainAxisStatus.q_xPowerFault	AND xPowerSupply01);

IF xPowerSupply02 THEN
	fbPwr02Fault(i_xConditions := stMasterModule.iq_astSubModuleAxis[CST_MasterPowerSupply02].iq_stStatus.q_stMainAxisStatus.q_xPowerFault	AND xPowerSupply02);
END_IF

(* Bleeder fault alarms *)
fbPwr01BleederFault(i_xConditions := stMasterModule.iq_astSubModuleAxis[CST_MasterPowerSupply01].iq_stStatus.q_stMainAxisStatus.q_xBleederFault	AND xPowerSupply01);
IF xPowerSupply02 THEN
	fbPwr02BleederFault(i_xConditions := stMasterModule.iq_astSubModuleAxis[CST_MasterPowerSupply02].iq_stStatus.q_stMainAxisStatus.q_xBleederFault	AND xPowerSupply02);
END_IF

(* Master axis error *)
fbMasterError(i_xConditions := stMasterModule.iq_astSubModuleAxis[CST_MachineMasterAxis].iq_stStatus.q_stMainAxisStatus.q_xError);

(* Power supply error *)
fbPwr01Error(i_xConditions := stMasterModule.iq_astSubModuleAxis[CST_MasterPowerSupply01].iq_stStatus.q_stMainAxisStatus.q_xError);
IF xPowerSupply02 THEN
	fbPwr02Error(i_xConditions := stMasterModule.iq_astSubModuleAxis[CST_MasterPowerSupply02].iq_stStatus.q_stMainAxisStatus.q_xError);
END_IF
END_STEP
STEP Output:
(* Sub Module Status Informations *)
stMasterModule.iq_stStatus.q_xModulePowered			:= stMasterModule.iq_astSubModuleAxis[CST_MachineMasterAxis].iq_stStatus.q_stMainAxisStatus.q_xPoweredOn;
stMasterModule.iq_stStatus.q_xModuleStopped			:= stMasterModule.iq_astSubModuleAxis[CST_MachineMasterAxis].iq_stStatus.q_stMainAxisStatus.q_xStopped;
stMasterModule.iq_stStatus.q_xModuleSynchronized	:= stMasterModule.iq_astSubModuleAxis[CST_MachineMasterAxis].iq_stStatus.q_stMainAxisStatus.q_xSynchronized;

(*Modalities Bits *)
stMasterModule.iq_stStatus.q_xNoOpActive			:= xNoOpActive;
stMasterModule.iq_stStatus.q_xAutoActive 			:= xAutoActive;
stMasterModule.iq_stStatus.q_xPositioningActive 	:= xPositioningActive;
stMasterModule.iq_stStatus.q_xJogActive		 		:= xJogActive;
stMasterModule.iq_stStatus.q_xCombiActive			:= xCombiActive;
stMasterModule.iq_stStatus.q_xCombiSynchroStopDone	:= xCombiSynchroStopDone;

IF NOT stMasterModule.iq_stCmd.i_xMasterRephasingRequest AND stMasterModule.iq_stStatus.q_xMasterRephased THEN
	stMasterModule.iq_stStatus.q_xMasterRephased 	:= FALSE;
END_IF

stMasterModule.iq_stStatus.q_xInitDone	:= (stMasterModule.iq_astSubModuleAxis[CST_MasterPowerSupply01].iq_stStatus.q_stMainAxisStatus.q_xInitDone OR NOT xPowerSupply01) AND
											(stMasterModule.iq_astSubModuleAxis[CST_MasterPowerSupply01].iq_stStatus.q_stMainAxisStatus.q_xInitDone OR NOT xPowerSupply02);
END_STEP
TRANSITION FROM (Input,SubModuleCalls,SetException,Output) TO Init:=
FALSE
END_TRANSITION
(* @SFCISJUMP := 'Init' *)
END_PROGRAM
```

#### Init.st - Init code
```iecst
PROGRAM _INIT
	stMasterModule ACCESS ADR(VAR_Machine.stMasterModule);
	stMasterModule.iq_stStatus.q_xAlarmXCoreEnabled	:= FALSE;

	IF VAR_AxPowerSupply01.nc_obj_inf.node_nr > 0 THEN
		xPowerSupply01	:= TRUE;
	END_IF

	IF VAR_AxPowerSupply02.nc_obj_inf.node_nr > 0 THEN
		xPowerSupply02	:= TRUE;
	END_IF
END_PROGRAM
```

#### Variables.var - Local variables
```iecst
(*Initialization*)
VAR
	xCpuInitDone : BOOL;
END_VAR
(* Input Variables *)
VAR
	xInputAuto : BOOL;
	xInputJog : BOOL;
	xInputCombi : BOOL;
	xInputPositioning : BOOL;
	xInputSelHoming : BOOL;
END_VAR
(*Modality Bits*)
VAR
	xModeReady : BOOL;
	xExitStep : BOOL; (*Exit Step Variables*)
	xAutoMode : BOOL; (*Auto Mode Command Variables*)
	xJogMode : BOOL; (*Jog Mode Command Variables*)
	xCombiMode : BOOL; (*Combi Mode Command Variables*)
	xPositioningMode : BOOL; (*Positioning Mode Command Variable*)
	xSelectiveHomeMode : BOOL;
END_VAR
(*Axes Enabling*)
VAR
	xPowerSupply01 : BOOL;
	xPowerSupply02 : BOOL;
END_VAR
(*FB Declarations*)
VAR
	fbPowerSupply01 : FB_GeneralAxis;
	fbPowerSupply02 : FB_GeneralAxis;
	fbMachineMasterSlow : FB_GeneralAxis; (*V4.A.A.1.6.10*)
END_VAR
(*Local Module Struct*)
VAR
	stMasterModule : REFERENCE TO ST_MasterModuleInterface; (*Master Module Interface Variables*)
	fbMpAlarmXCore : MpAlarmXCore;
END_VAR
(*FB Alarms*)
VAR
	fbMasterError : FB_ExceptionAlarmX;
	fbPwr01Error : FB_ExceptionAlarmX;
	fbPwr02Error : FB_ExceptionAlarmX;
	fbPwr01Fault : FB_ExceptionAlarmX;
	fbPwr02Fault : FB_ExceptionAlarmX;
	fbPwr01BleederFault : FB_ExceptionAlarmX;
	fbPwr02BleederFault : FB_ExceptionAlarmX;
END_VAR
(*Local Variables*)
VAR
	xReactionActive : BOOL; (*Quick stop, emergency stop or shutdown requested to Master module*)
	uiAxisIndex : UINT; (*Axis Index*)
	uiAxisToken : UINT;
	uiNumberOfSteps : UINT;
	rAxisDistance : REAL;
	tofReactionActive : TOF;
END_VAR
(*Active Modality Bits*)
VAR
	xNoOpActive : BOOL;
	xAutoActive : BOOL;
	xPositioningActive : BOOL;
	xCombiActive : BOOL;
	xJogActive : BOOL;
	xSelHomingActive : BOOL;
	xCombiSynchroStopDone : BOOL;
END_VAR
(*Sequencer Steps*)
VAR
	uiPositioningStep : UINT;
	uiAutoStep : UINT;
	uiJogStep : UINT;
	uiCombiStep : UINT;
	uiSelectiveHomeStep : UINT;
END_VAR
```

### Program Logical/30_MC/Task/Cyclic02/MC_FILLER (IEC) - MC_FILLER - C#1 0.8ms or C#2 10.4ms

#### Variables.var
```iecst
(* Input Variables *)
VAR
	xInputAuto : BOOL;
	xInputVelocity : BOOL;
	xInputJogMulti : BOOL;
	xInputAutoMulti : BOOL;
	xInputSelHoming : BOOL;
	xInputThirdPartySetup : BOOL;
	xInputInductionSetup : BOOL;
	xInputPositioning : BOOL;
	xInputSlowMotion : BOOL;
	xInputBrakeRelease : BOOL;
	xInputStepByStepSingleAxis : BOOL; (*V4.A.A.1.7.0*)
	xInputStepByStep : BOOL;
END_VAR
(*Modality Bits*)
VAR
	xModeReady : BOOL;
	xExitStep : BOOL; (*Exit Step Variables*)
	xAutoMode : BOOL; (*Auto Mode Command Variables*)
	xVelocityMode : BOOL; (*Positioning Mode Command Variable*)
	xPositioningMode : BOOL; (*Positioning Mode Command Variable*)
	xThirdPartySetupMode : BOOL;
	xInductionSetupMode : BOOL;
	xSelectiveHomingMode : BOOL; (*Selective Homing Command Variable*)
	xBrakeReleaseMode : BOOL;
	xAutoMultiMode : BOOL;
	xJogMultiMode : BOOL;
	xStepByStepMode : BOOL;
	xSlowMotionMode : BOOL;
	xModulePowered : BOOL;
	xRealAxesReadyForACommand : BOOL;
	xSynchroWithOffset : BOOL;
	xModuleStopped : BOOL;
	xRealAxesSynchronized : BOOL;
	xPhaseShiftDone : BOOL;
	xSelHomingDone : BOOL;
	xModuleInitialized : BOOL;
	xModuleHomed : BOOL;
END_VAR
(*Active Modality Bits*)
VAR
	xNoOpActive : BOOL;
	xAutoActive : BOOL;
	xPositioningActive : BOOL;
	xThirdPartySetupActive : BOOL;
	xInductionSetupActive : BOOL;
	xSelHomingActive : BOOL;
	xBrakeReleaseActive : BOOL;
	xVelocityActive : BOOL;
	xSlowMotionActive : BOOL;
	xJogMultiActive : BOOL;
	xAutoMultiActive : BOOL;
	xStepByStepActive : BOOL;
END_VAR
(*Axes presence*)
VAR
	axAxisPresent : ARRAY[CST_FirstFillerModuleAxis..CST_LastFillerModuleAxis] OF BOOL := [17(FALSE)];
END_VAR
(*Local master management*)
VAR
	usiMasterRequest : E_MasterStatus;
	usiMasterStatus : E_MasterStatus;
	usiMasterTempStatus : E_MasterStatus;
END_VAR
(*FB axis Declarations*)
VAR
	fbFillerMaster : FB_GeneralAxis;
	fbMain : FB_GeneralAxis;
	fbInlet01 : FB_GeneralAxis;
	fbInlet02 : FB_GeneralAxis;
	fbInlet03 : FB_GeneralAxis;
	fbInlet04 : FB_GeneralAxis;
	fbInlet05 : FB_GeneralAxis;
	fbInlet06 : FB_GeneralAxis;
	fbInlet07 : FB_GeneralAxis;
	fbInlet08 : FB_GeneralAxis;
	fbInlet09 : FB_GeneralAxis;
	fbInlet10 : FB_GeneralAxis;
	fbOutlet01 : FB_GeneralAxis;
	fbOutlet02 : FB_GeneralAxis;
	fbOutlet03 : FB_GeneralAxis;
	fbOutlet04 : FB_GeneralAxis;
	fbOutlet05 : FB_GeneralAxis;
	fbOutlet06 : FB_GeneralAxis;
END_VAR
(*Local Module Struct*)
VAR
	stFillerModule : REFERENCE TO ST_FillerModuleInterface; (*Filler Module Interface Variables*)
	fbMpAlarmXCore : MpAlarmXCore;
END_VAR
(*FB Alarms*)
VAR
	fbQuickStopFromPlc : FB_ExceptionAlarmX;
	fbMainAxisLagError : FB_ExceptionAlarmX;
	fbInlet01LagError : FB_ExceptionAlarmX;
	fbInlet02LagError : FB_ExceptionAlarmX;
	fbInlet03LagError : FB_ExceptionAlarmX;
	fbInlet04LagError : FB_ExceptionAlarmX;
	fbInlet05LagError : FB_ExceptionAlarmX;
	fbInlet06LagError : FB_ExceptionAlarmX;
	fbInlet07LagError : FB_ExceptionAlarmX;
	fbInlet08LagError : FB_ExceptionAlarmX;
	fbInlet09LagError : FB_ExceptionAlarmX;
	fbInlet10LagError : FB_ExceptionAlarmX;
	fbOutlet01LagError : FB_ExceptionAlarmX;
	fbOutlet02LagError : FB_ExceptionAlarmX;
	fbOutlet03LagError : FB_ExceptionAlarmX;
	fbOutlet04LagError : FB_ExceptionAlarmX;
	fbOutlet05LagError : FB_ExceptionAlarmX;
	fbOutlet06LagError : FB_ExceptionAlarmX;
	fbEmergencyStopAlarm : FB_ExceptionAlarmX;
	fbMasterError : FB_ExceptionAlarmX;
	fbMainAxisError : FB_ExceptionAlarmX;
	fbInlet01Error : FB_ExceptionAlarmX;
	fbInlet02Error : FB_ExceptionAlarmX;
	fbInlet03Error : FB_ExceptionAlarmX;
	fbInlet04Error : FB_ExceptionAlarmX;
	fbInlet05Error : FB_ExceptionAlarmX;
	fbInlet06Error : FB_ExceptionAlarmX;
	fbInlet07Error : FB_ExceptionAlarmX;
	fbInlet08Error : FB_ExceptionAlarmX;
	fbInlet09Error : FB_ExceptionAlarmX;
	fbInlet10Error : FB_ExceptionAlarmX;
	fbOutlet01Error : FB_ExceptionAlarmX;
	fbOutlet02Error : FB_ExceptionAlarmX;
	fbOutlet03Error : FB_ExceptionAlarmX;
	fbOutlet04Error : FB_ExceptionAlarmX;
	fbOutlet05Error : FB_ExceptionAlarmX;
	fbOutlet06Error : FB_ExceptionAlarmX;
END_VAR
(*Local Variables*)
VAR
	xFillerPositionValid : BOOL; (*//V4.A.A.1.6.12e*)
	xRinserPositionValid : BOOL; (*//V4.A.A.1.6.12e*)
	xCapperPositionValid : BOOL; (*//V4.A.A.1.6.12e*)
	xCrownerPositionValid : BOOL; (*//V4.A.A.1.6.12e*)
	xDoserPositionValid : BOOL; (*//V4.A.A.1.6.12e*)
	xReactionActive : BOOL;
	xParityPhase : BOOL;
	iTempParity : INT;
	lrTempOldPosition : LREAL;
	lrTempPosDiff : LREAL;
	uiAxisIndex : UINT; (*Axis Index*)
	uiOldAxisSelected : UINT;
	uiNextHomingPositionIndex : UINT; (*Temp var for initializing homing position chain*)
	uiFirstFillerModuleAxis : UINT; (*First axis index in filler module*)
	uiLastFillerModuleAxis : UINT; (*Last axis index in filler module*)
	uiAxisToken : UINT;
	uiNumberOfSteps : UINT;
	uiSlowAxisIndex : UINT;
	rModuleVelocity : REAL;
	rAxisDistance : REAL;
	lrFillerAbsolutePosition : LREAL; (*//V4.A.A.1.6.12e*)
	lrRinserAbsolutePosition : LREAL; (*//V4.A.A.1.6.12e*)
	lrCapperAbsolutePosition : LREAL; (*//V4.A.A.1.6.12e*)
	lrCrownerAbsolutePosition : LREAL; (*//V4.A.A.1.6.12e*)
	lrDoserAbsolutePosition : LREAL; (*//V4.A.A.1.6.12e*)
	lrIncrement : LREAL;
	lrOldPosition : LREAL;
	tonPositDone : TON;
	tofReactionActive : TOF;
	axPresentIndex : USINT;
END_VAR
(*Sequencer Steps*)
VAR
	uiVelocityStep : UINT;
	uiAutoStep : UINT;
	uiPositioningStep : UINT;
	uiThirdPartySetupStep : UINT;
	uiInductionSetupStep : UINT;
	uiSelectiveHomeStep : UINT;
	uiBrakeReleaseStep : UINT;
	uiSlowMotionStep : UINT;
	uiJogMulti : UINT;
	uiAutoMulti : UINT;
	uiStepByStep : UINT;
	auiAxisTokenList : ARRAY[0..20] OF UINT;
	uiTokenIndex : UINT;
END_VAR
(*Absolute Position Calculation FBs*)
(*//V4.A.A.1.6.12e*)
VAR
	fbFillerAbsPos : FB_AbsolutePosCalculation; (*//V4.A.A.1.6.12e*)
	fbRinserAbsPos : FB_AbsolutePosCalculation; (*//V4.A.A.1.6.12e*)
	fbCapperAbsPos : FB_AbsolutePosCalculation; (*//V4.A.A.1.6.12e*)
	fbCrownerAbsPos : FB_AbsolutePosCalculation; (*//V4.A.A.1.6.12e*)
	fbDoserAbsPos : FB_AbsolutePosCalculation; (*//V4.A.A.1.6.12e*)
END_VAR
```
